C07295=1233.032,115.078,-48.574,-178.231,5.533,148.437
C07296=1233.037,114.829,-48.555,-178.233,5.532,148.437
C07297=1233.042,114.580,-48.535,-178.236,5.532,148.438
C07298=1233.046,114.331,-48.516,-178.239,5.530,148.438
C07299=1233.051,114.082,-48.497,-178.241,5.529,148.439
C07300=1233.056,113.832,-48.477,-178.244,5.529,148.439
C07301=1233.062,113.583,-48.458,-178.246,5.528,148.440
C07302=1233.066,113.334,-48.438,-178.248,5.527,148.441
C07303=1233.070,113.084,-48.419,-178.251,5.526,148.441
C07304=1233.075,112.836,-48.399,-178.254,5.525,148.442
C07305=1233.080,112.587,-48.380,-178.256,5.524,148.442
C07306=1233.085,112.337,-48.360,-178.259,5.524,148.443
C07307=1233.090,112.088,-48.341,-178.261,5.523,148.443
C07308=1233.094,111.839,-48.322,-178.264,5.521,148.444
C07309=1233.099,111.590,-48.302,-178.267,5.520,148.445
C07310=1233.104,111.341,-48.283,-178.269,5.520,148.445
C07311=1233.109,111.091,-48.263,-178.271,5.519,148.446
C07312=1233.114,110.842,-48.244,-178.274,5.518,148.446
C07313=1233.118,110.593,-48.225,-178.277,5.516,148.447
C07314=1233.124,110.344,-48.205,-178.279,5.516,148.447
C07315=1233.128,110.094,-48.186,-178.282,5.515,148.448
C07316=1233.132,109.845,-48.167,-178.284,5.514,148.448
C07317=1233.138,109.596,-48.147,-178.287,5.514,148.449
C07318=1233.143,109.347,-48.128,-178.289,5.513,148.450
C07319=1233.147,109.098,-48.110,-178.292,5.511,148.450
C07320=1233.152,108.848,-48.090,-178.295,5.511,148.451
C07321=1233.157,108.599,-48.071,-178.297,5.510,148.451
C07322=1233.162,108.350,-48.052,-178.299,5.509,148.452
C07323=1233.166,108.081,-48.031,-178.302,5.508,148.452
C07324=1233.172,107.813,-48.010,-178.305,5.507,148.453
C07325=1233.177,107.545,-47.989,-178.308,5.506,148.454
C07326=1233.183,107.276,-47.969,-178.310,5.506,148.454
C07327=1233.187,107.026,-47.949,-178.313,5.504,148.455
C07328=1233.192,106.778,-47.930,-178.316,5.503,148.455
C07329=1233.197,106.528,-47.911,-178.318,5.503,148.456
C07330=1233.201,106.280,-47.892,-178.320,5.502,148.456
C07331=1233.206,106.030,-47.873,-178.323,5.501,148.457
C07332=1233.212,105.781,-47.854,-178.326,5.500,148.458
C07333=1233.216,105.531,-47.835,-178.329,5.499,148.458
C07334=1233.221,105.283,-47.815,-178.331,5.498,148.459
C07335=1233.226,105.033,-47.796,-178.334,5.497,148.459
C07336=1233.231,104.784,-47.778,-178.336,5.497,148.460
C07337=1233.236,104.534,-47.758,-178.338,5.496,148.460
C07338=1233.240,104.286,-47.739,-178.341,5.495,148.461
C07339=1233.245,104.036,-47.720,-178.344,5.495,148.462
C07340=1233.250,103.787,-47.702,-178.346,5.493,148.462
C07341=1233.255,103.537,-47.682,-178.349,5.492,148.463
C07342=1233.260,103.289,-47.663,-178.351,5.491,148.463
C07343=1233.264,103.039,-47.644,-178.354,5.491,148.464
C07344=1233.270,102.790,-47.625,-178.356,5.490,148.464
C07345=1233.274,102.541,-47.606,-178.359,5.489,148.465
C07346=1233.279,102.292,-47.587,-178.361,5.489,148.466
C07347=1233.283,102.042,-47.569,-178.364,5.487,148.466
C07348=1233.289,101.793,-47.549,-178.367,5.486,148.467
C07349=1233.293,101.544,-47.530,-178.369,5.486,148.467
C07350=1233.298,101.294,-47.512,-178.371,5.485,148.468
C07351=1233.303,101.046,-47.493,-178.374,5.484,148.469
C07352=1233.308,100.796,-47.473,-178.377,5.483,148.469
C07353=1233.312,100.547,-47.455,-178.379,5.482,148.470
C07354=1233.317,100.297,-47.436,-178.382,5.481,148.470
C07355=1233.322,100.049,-47.417,-178.385,5.480,148.471
C07356=1233.327,99.799,-47.398,-178.387,5.480,148.472
C07357=1233.331,99.550,-47.379,-178.389,5.479,148.472
C07358=1233.336,99.301,-47.361,-178.392,5.478,148.473
C07359=1233.341,99.051,-47.342,-178.395,5.478,148.473
C07360=1233.346,98.803,-47.323,-178.397,5.477,148.474
C07361=1233.351,98.553,-47.304,-178.399,5.476,148.474
C07362=1233.355,98.304,-47.285,-178.402,5.475,148.475
C07363=1233.361,98.055,-47.267,-178.405,5.474,148.476
C07364=1233.365,97.805,-47.248,-178.407,5.473,148.476
C07365=1233.370,97.556,-47.230,-178.410,5.472,148.477
C07366=1233.375,97.307,-47.210,-178.412,5.472,148.477
C07367=1233.380,97.057,-47.192,-178.415,5.471,148.478
C07368=1233.385,96.808,-47.173,-178.417,5.470,148.478
C07369=1233.389,96.559,-47.154,-178.420,5.470,148.479
C07370=1233.394,96.310,-47.136,-178.422,5.469,148.480
C07371=1233.399,96.061,-47.117,-178.425,5.467,148.480
C07372=1233.403,95.811,-47.098,-178.428,5.467,148.481
C07373=1233.409,95.562,-47.080,-178.430,5.466,148.481
C07374=1233.413,95.313,-47.060,-178.433,5.465,148.482
C07375=1233.418,95.063,-47.042,-178.435,5.464,148.482
C07376=1233.424,94.814,-47.024,-178.438,5.464,148.483
C07377=1233.428,94.565,-47.005,-178.440,5.463,148.484
C07378=1233.433,94.315,-46.987,-178.443,5.463,148.484
C07379=1233.438,94.067,-46.968,-178.445,5.462,148.485
C07380=1233.442,93.817,-46.949,-178.448,5.461,148.485
C07381=1233.447,93.568,-46.931,-178.450,5.460,148.486
C07382=1233.453,93.319,-46.912,-178.454,5.459,148.487
C07383=1233.457,93.069,-46.894,-178.456,5.458,148.487
C07384=1233.461,92.820,-46.875,-178.458,5.457,148.488
C07385=1233.466,92.571,-46.857,-178.461,5.457,148.488
C07386=1233.472,92.322,-46.838,-178.463,5.456,148.489
C07387=1233.476,92.072,-46.819,-178.466,5.455,148.490
C07388=1233.481,91.823,-46.801,-178.468,5.455,148.490
C07389=1233.487,91.574,-46.783,-178.471,5.454,148.491
C07390=1233.491,91.324,-46.764,-178.473,5.453,148.491
C07391=1233.495,91.075,-46.746,-178.476,5.452,148.492
C07392=1233.500,90.826,-46.728,-178.478,5.452,148.493
C07393=1233.506,90.577,-46.709,-178.481,5.451,148.493
C07394=1233.510,90.327,-46.690,-178.484,5.450,148.494
C07395=1233.515,90.078,-46.672,-178.486,5.449,148.494
C07396=1233.520,89.829,-46.654,-178.489,5.448,148.495
C07397=1233.524,89.579,-46.636,-178.491,5.448,148.496
C07398=1233.530,89.330,-46.617,-178.494,5.447,148.496
C07399=1233.534,89.081,-46.599,-178.496,5.446,148.497
C07400=1233.539,88.832,-46.581,-178.499,5.445,148.497
C07401=1233.544,88.582,-46.562,-178.501,5.445,148.498
C07402=1233.549,88.333,-46.544,-178.504,5.444,148.499
C07403=1233.554,88.084,-46.525,-178.506,5.443,148.499
C07404=1233.559,87.835,-46.507,-178.509,5.443,148.500
C07405=1233.563,87.585,-46.489,-178.511,5.442,148.500
C07406=1233.568,87.336,-46.471,-178.514,5.441,148.501
C07407=1233.573,87.087,-46.453,-178.516,5.440,148.501
C07408=1233.578,86.837,-46.435,-178.519,5.440,148.502
C07409=1233.583,86.589,-46.415,-178.522,5.438,148.503
C07410=1233.588,86.339,-46.397,-178.525,5.438,148.503
C07411=1233.592,86.089,-46.379,-178.527,5.437,148.504
C07412=1233.597,85.840,-46.361,-178.529,5.436,148.504
C07413=1233.602,85.591,-46.343,-178.532,5.436,148.505
C07414=1233.607,85.342,-46.325,-178.535,5.435,148.506
C07415=1233.612,85.092,-46.307,-178.537,5.434,148.506
C07416=1233.616,84.843,-46.289,-178.539,5.433,148.507
C07417=1233.621,84.594,-46.271,-178.542,5.433,148.508
C07418=1233.627,84.344,-46.252,-178.545,5.432,148.508
C07419=1233.632,84.095,-46.234,-178.547,5.432,148.509
C07420=1233.636,83.846,-46.215,-178.550,5.431,148.509
C07421=1233.641,83.597,-46.197,-178.552,5.430,148.510
C07422=1233.646,83.347,-46.179,-178.555,5.429,148.511
C07423=1233.651,83.098,-46.161,-178.557,5.429,148.511
C07424=1233.656,82.849,-46.143,-178.560,5.428,148.512
C07425=1233.660,82.600,-46.125,-178.562,5.427,148.512
C07426=1233.665,82.350,-46.107,-178.565,5.427,148.513
C07427=1233.670,82.082,-46.088,-178.568,5.425,148.514
C07428=1233.675,81.813,-46.069,-178.570,5.425,148.514
C07429=1233.681,81.544,-46.049,-178.573,5.424,148.515
C07430=1233.686,81.276,-46.029,-178.576,5.423,148.516
C07431=1233.691,81.027,-46.011,-178.578,5.423,148.516
C07432=1233.696,80.778,-45.993,-178.581,5.422,148.517
C07433=1233.701,80.529,-45.975,-178.584,5.422,148.518
C07434=1233.706,80.279,-45.958,-178.586,5.421,148.518
C07435=1233.711,80.030,-45.940,-178.588,5.420,148.519
C07436=1233.716,79.781,-45.922,-178.591,5.420,148.519
C07437=1233.721,79.532,-45.904,-178.594,5.419,148.520
C07438=1233.726,79.282,-45.886,-178.596,5.418,148.521
C07439=1233.730,79.032,-45.868,-178.599,5.418,148.521
C07440=1233.735,78.783,-45.850,-178.601,5.417,148.522
C07441=1233.739,78.534,-45.833,-178.604,5.416,148.522
C07442=1233.744,78.285,-45.815,-178.606,5.416,148.523
C07443=1233.749,78.036,-45.797,-178.609,5.415,148.524
C07444=1233.754,77.787,-45.779,-178.611,5.414,148.524
C07445=1233.759,77.537,-45.761,-178.614,5.413,148.525
C07446=1233.764,77.288,-45.743,-178.616,5.413,148.525
C07447=1233.769,77.038,-45.725,-178.619,5.412,148.526
C07448=1233.774,76.789,-45.707,-178.621,5.412,148.527
C07449=1233.779,76.540,-45.689,-178.624,5.411,148.527
C07450=1233.784,76.290,-45.672,-178.626,5.410,148.528
C07451=1233.789,76.041,-45.654,-178.629,5.409,148.528
C07452=1233.793,75.791,-45.636,-178.631,5.409,148.529
C07453=1233.797,75.542,-45.618,-178.634,5.408,148.530
C07454=1233.803,75.293,-45.601,-178.637,5.408,148.530
C07455=1233.807,75.043,-45.583,-178.639,5.407,148.531
C07456=1233.812,74.794,-45.565,-178.641,5.406,148.532
C07457=1233.817,74.545,-45.547,-178.644,5.406,148.532
C07458=1233.823,74.295,-45.530,-178.647,5.405,148.533
C07459=1233.827,74.046,-45.512,-178.649,5.404,148.534
C07460=1233.832,73.797,-45.495,-178.652,5.404,148.534
C07461=1233.837,73.547,-45.477,-178.654,5.403,148.535
C07462=1233.842,73.298,-45.459,-178.657,5.402,148.535
C07463=1233.847,73.049,-45.441,-178.659,5.402,148.536
C07464=1233.852,72.799,-45.424,-178.662,5.401,148.537
C07465=1233.856,72.550,-45.407,-178.665,5.400,148.537
C07466=1233.861,72.301,-45.389,-178.667,5.400,148.538
C07467=1233.866,72.051,-45.372,-178.669,5.399,148.538
C07468=1233.871,71.802,-45.354,-178.672,5.398,148.539
C07469=1233.876,71.553,-45.336,-178.675,5.398,148.540
C07470=1233.880,71.304,-45.319,-178.677,5.397,148.540
C07471=1233.885,71.054,-45.301,-178.680,5.397,148.541
C07472=1233.891,70.805,-45.284,-178.683,5.396,148.542
C07473=1233.896,70.555,-45.266,-178.685,5.395,148.542
C07474=1233.900,70.306,-45.248,-178.687,5.394,148.543
C07475=1233.905,70.057,-45.231,-178.690,5.394,148.543
C07476=1233.910,69.808,-45.213,-178.693,5.393,148.544
C07477=1233.915,69.558,-45.196,-178.695,5.393,148.545
C07478=1233.919,69.309,-45.178,-178.698,5.392,148.545
C07479=1233.925,69.060,-45.162,-178.700,5.391,148.546
C07480=1233.930,68.811,-45.144,-178.703,5.390,148.546
C07481=1233.935,68.561,-45.126,-178.705,5.390,148.547
C07482=1233.939,68.312,-45.109,-178.708,5.389,148.548
C07483=1233.945,68.062,-45.092,-178.710,5.389,148.548
C07484=1233.949,67.813,-45.074,-178.713,5.388,148.549
C07485=1233.954,67.564,-45.057,-178.716,5.388,148.550
C07486=1233.959,67.314,-45.039,-178.718,5.387,148.550
C07487=1233.964,67.065,-45.022,-178.721,5.386,148.551
C07488=1233.968,66.816,-45.004,-178.723,5.385,148.552
C07489=1233.973,66.566,-44.987,-178.726,5.385,148.552
C07490=1233.978,66.317,-44.969,-178.728,5.384,148.553
C07491=1233.983,66.067,-44.952,-178.731,5.384,148.554
C07492=1233.988,65.819,-44.935,-178.734,5.383,148.554
C07493=1233.994,65.569,-44.918,-178.736,5.382,148.555
C07494=1233.998,65.320,-44.901,-178.738,5.382,148.555
C07495=1234.003,65.070,-44.883,-178.741,5.381,148.556
C07496=1234.008,64.821,-44.866,-178.743,5.381,148.557
C07497=1234.012,64.572,-44.848,-178.746,5.381,148.557
C07498=1234.018,64.322,-44.831,-178.748,5.380,148.558
C07499=1234.022,64.072,-44.814,-178.751,5.379,148.559
C07500=1234.027,63.823,-44.796,-178.754,5.379,148.559
C07501=1234.033,63.574,-44.779,-178.756,5.378,148.560
C07502=1234.037,63.325,-44.763,-178.758,5.377,148.560
C07503=1234.042,63.076,-44.745,-178.761,5.377,148.561
C07504=1234.047,62.826,-44.728,-178.764,5.376,148.562
C07505=1234.052,62.576,-44.711,-178.766,5.376,148.562
C07506=1234.057,62.327,-44.693,-178.769,5.375,148.563
C07507=1234.061,62.078,-44.676,-178.772,5.374,148.564
C07508=1234.067,61.828,-44.659,-178.774,5.374,148.564
C07509=1234.071,61.580,-44.642,-178.776,5.373,148.565
C07510=1234.077,61.330,-44.625,-178.779,5.372,148.565
C07511=1234.081,61.080,-44.608,-178.782,5.372,148.566
C07512=1234.086,60.831,-44.591,-178.784,5.371,148.567
C07513=1234.090,60.582,-44.573,-178.786,5.371,148.567
C07514=1234.096,60.333,-44.556,-178.789,5.371,148.568
C07515=1234.101,60.083,-44.540,-178.792,5.370,148.569
C07516=1234.106,59.833,-44.523,-178.794,5.370,148.569
C07517=1234.110,59.584,-44.505,-178.796,5.369,148.570
C07518=1234.115,59.335,-44.488,-178.799,5.368,148.571
C07519=1234.120,59.086,-44.472,-178.802,5.367,148.571
C07520=1234.126,58.836,-44.454,-178.804,5.367,148.572
C07521=1234.130,58.587,-44.438,-178.807,5.366,148.573
C07522=1234.135,58.337,-44.420,-178.810,5.366,148.573
C07523=1234.139,58.088,-44.403,-178.812,5.365,148.574
C07524=1234.145,57.839,-44.386,-178.815,5.365,148.575
C07525=1234.150,57.589,-44.369,-178.817,5.364,148.575
C07526=1234.155,57.340,-44.352,-178.819,5.364,148.576
C07527=1234.159,57.090,-44.335,-178.822,5.363,148.576
C07528=1234.165,56.841,-44.319,-178.824,5.363,148.577
C07529=1234.169,56.592,-44.301,-178.827,5.362,148.578
C07530=1234.174,56.343,-44.285,-178.830,5.361,148.578
C07531=1234.180,56.074,-44.266,-178.832,5.361,148.579
C07532=1234.185,55.806,-44.248,-178.835,5.360,148.580
C07533=1234.190,55.536,-44.230,-178.837,5.360,148.580
C07534=1234.196,55.269,-44.212,-178.840,5.359,148.581
C07535=1234.201,55.019,-44.195,-178.843,5.359,148.582
C07536=1234.205,54.770,-44.178,-178.845,5.358,148.582
C07537=1234.211,54.521,-44.161,-178.848,5.357,148.583
C07538=1234.215,54.271,-44.144,-178.851,5.357,148.584
C07539=1234.220,54.022,-44.128,-178.853,5.356,148.584
C07540=1234.226,53.773,-44.111,-178.856,5.356,148.585
C07541=1234.230,53.523,-44.094,-178.859,5.355,148.586
C07542=1234.234,53.274,-44.077,-178.861,5.355,148.586
C07543=1234.240,53.024,-44.060,-178.864,5.354,148.587
C07544=1234.245,52.775,-44.044,-178.865,5.354,148.587
C07545=1234.249,52.526,-44.027,-178.868,5.353,148.588
C07546=1234.254,52.276,-44.010,-178.871,5.353,148.589
C07547=1234.260,52.027,-43.993,-178.873,5.352,148.589
C07548=1234.264,51.778,-43.977,-178.876,5.352,148.590
C07549=1234.269,51.528,-43.960,-178.879,5.351,148.591
C07550=1234.275,51.278,-43.944,-178.881,5.350,148.591
C07551=1234.279,51.029,-43.927,-178.884,5.350,148.592
C07552=1234.284,50.779,-43.910,-178.886,5.349,148.593
C07553=1234.289,50.530,-43.894,-178.889,5.349,148.594
C07554=1234.294,50.281,-43.877,-178.891,5.349,148.594
C07555=1234.298,50.031,-43.860,-178.893,5.348,148.595
C07556=1234.304,49.782,-43.843,-178.896,5.347,148.595
C07557=1234.309,49.533,-43.827,-178.899,5.347,148.596
C07558=1234.313,49.283,-43.810,-178.901,5.346,148.597
C07559=1234.319,49.034,-43.793,-178.904,5.346,148.597
C07560=1234.324,48.784,-43.777,-178.906,5.345,148.598
C07561=1234.328,48.535,-43.761,-178.909,5.345,148.599
C07562=1234.333,48.286,-43.744,-178.911,5.345,148.599
C07563=1234.338,48.036,-43.728,-178.914,5.344,148.600
C07564=1234.343,47.787,-43.710,-178.916,5.344,148.601
C07565=1234.348,47.538,-43.694,-178.919,5.343,148.601
C07566=1234.353,47.288,-43.678,-178.922,5.342,148.602
C07567=1234.358,47.039,-43.662,-178.924,5.342,148.603
C07568=1234.363,46.789,-43.645,-178.927,5.341,148.603
C07569=1234.368,46.540,-43.628,-178.929,5.340,148.604
C07570=1234.373,46.291,-43.612,-178.931,5.341,148.604
C07571=1234.378,46.041,-43.596,-178.934,5.340,148.605
C07572=1234.383,45.792,-43.579,-178.937,5.339,148.606
C07573=1234.388,45.542,-43.562,-178.939,5.339,148.606
C07574=1234.392,45.293,-43.545,-178.942,5.338,148.607
C07575=1234.398,45.043,-43.530,-178.944,5.338,148.608
C07576=1234.402,44.794,-43.513,-178.947,5.337,148.608
C07577=1234.407,44.545,-43.497,-178.949,5.337,148.609
C07578=1234.412,44.296,-43.480,-178.952,5.337,148.610
C07579=1234.417,44.045,-43.464,-178.954,5.336,148.611
C07580=1234.422,43.796,-43.447,-178.957,5.336,148.611
C07581=1234.427,43.547,-43.431,-178.960,5.335,148.612
C07582=1234.432,43.297,-43.415,-178.962,5.334,148.612
C07583=1234.437,43.048,-43.398,-178.964,5.334,148.613
C07584=1234.442,42.799,-43.382,-178.967,5.334,148.614
C07585=1234.447,42.549,-43.366,-178.969,5.333,148.614
C07586=1234.452,42.300,-43.350,-178.972,5.333,148.615
C07587=1234.456,42.051,-43.333,-178.974,5.332,148.616
C07588=1234.462,41.800,-43.317,-178.977,5.332,148.616
C07589=1234.467,41.552,-43.300,-178.980,5.331,148.617
C07590=1234.471,41.302,-43.284,-178.982,5.331,148.618
C07591=1234.477,41.053,-43.268,-178.984,5.331,148.618
C07592=1234.481,40.803,-43.251,-178.987,5.330,148.619
C07593=1234.486,40.554,-43.236,-178.990,5.330,148.620
C07594=1234.491,40.304,-43.219,-178.992,5.329,148.620
C07595=1234.496,40.055,-43.204,-178.995,5.328,148.621
C07596=1234.501,39.805,-43.187,-178.998,5.328,148.622
C07597=1234.506,39.557,-43.171,-179.000,5.328,148.622
C07598=1234.511,39.307,-43.155,-179.002,5.328,148.623
C07599=1234.516,39.058,-43.138,-179.005,5.327,148.624
C07600=1234.521,38.808,-43.122,-179.007,5.326,148.624
C07601=1234.526,38.559,-43.106,-179.010,5.326,148.625
C07602=1234.530,38.309,-43.090,-179.012,5.325,148.626
C07603=1234.535,38.060,-43.074,-179.015,5.325,148.626
C07604=1234.540,37.810,-43.058,-179.017,5.325,148.627
C07605=1234.545,37.561,-43.042,-179.020,5.324,148.628
C07606=1234.550,37.311,-43.026,-179.022,5.324,148.628
C07607=1234.555,37.062,-43.009,-179.025,5.323,148.629
C07608=1234.560,36.812,-42.993,-179.028,5.322,148.630
C07609=1234.565,36.563,-42.977,-179.030,5.323,148.630
C07610=1234.570,36.314,-42.961,-179.032,5.322,148.631
C07611=1234.575,36.064,-42.945,-179.035,5.322,148.632
C07612=1234.580,35.815,-42.929,-179.038,5.321,148.632
C07613=1234.585,35.565,-42.913,-179.040,5.320,148.633
C07614=1234.590,35.316,-42.897,-179.043,5.320,148.634
C07615=1234.595,35.066,-42.881,-179.045,5.320,148.634
C07616=1234.600,34.817,-42.865,-179.048,5.320,148.635
C07617=1234.605,34.567,-42.849,-179.050,5.319,148.636
C07618=1234.610,34.318,-42.833,-179.053,5.318,148.636
C07619=1234.615,34.069,-42.817,-179.056,5.318,148.637
C07620=1234.620,33.819,-42.801,-179.058,5.317,148.638
C07621=1234.625,33.570,-42.785,-179.060,5.318,148.638
C07622=1234.629,33.320,-42.769,-179.063,5.317,148.639
C07623=1234.635,33.071,-42.754,-179.066,5.316,148.640
C07624=1234.639,32.821,-42.737,-179.068,5.316,148.640
C07625=1234.644,32.572,-42.721,-179.070,5.315,148.641
C07626=1234.650,32.323,-42.706,-179.072,5.315,148.642
C07627=1234.655,32.073,-42.690,-179.075,5.315,148.642
C07628=1234.660,31.824,-42.673,-179.078,5.314,148.643
C07629=1234.665,31.574,-42.658,-179.080,5.314,148.644
C07630=1234.669,31.325,-42.643,-179.083,5.313,148.644
C07631=1234.674,31.076,-42.626,-179.085,5.313,148.645
C07632=1234.679,30.826,-42.610,-179.088,5.313,148.646
C07633=1234.684,30.576,-42.595,-179.090,5.312,148.646
C07634=1234.690,30.327,-42.579,-179.093,5.312,148.647
C07635=1234.695,30.058,-42.562,-179.096,5.311,148.648
C07636=1234.700,29.789,-42.545,-179.099,5.311,148.649
C07637=1234.705,29.521,-42.528,-179.101,5.310,148.649
C07638=1234.711,29.253,-42.511,-179.104,5.310,148.650
C07639=1234.715,29.003,-42.495,-179.106,5.310,148.651
C07640=1234.721,28.754,-42.479,-179.109,5.309,148.651
C07641=1234.726,28.504,-42.463,-179.111,5.309,148.652
C07642=1234.731,28.254,-42.447,-179.114,5.308,148.653
C07643=1234.735,28.005,-42.432,-179.117,5.308,148.653
C07644=1234.740,27.756,-42.416,-179.119,5.308,148.654
C07645=1234.745,27.506,-42.400,-179.122,5.307,148.655
C07646=1234.751,27.257,-42.385,-179.124,5.307,148.655
C07647=1234.755,27.008,-42.370,-179.127,5.306,148.656
C07648=1234.760,26.758,-42.354,-179.129,5.306,148.657
C07649=1234.765,26.508,-42.338,-179.132,5.306,148.657
C07650=1234.771,26.259,-42.323,-179.134,5.305,148.658
C07651=1234.775,26.010,-42.306,-179.137,5.305,148.659
C07652=1234.780,25.760,-42.291,-179.139,5.304,148.659
C07653=1234.785,25.511,-42.275,-179.142,5.304,148.660
C07654=1234.791,25.261,-42.260,-179.144,5.304,148.661
C07655=1234.795,25.012,-42.244,-179.147,5.303,148.662
C07656=1234.800,24.762,-42.229,-179.149,5.303,148.662
C07657=1234.806,24.513,-42.213,-179.152,5.302,148.663
C07658=1234.810,24.263,-42.198,-179.154,5.303,148.664
C07659=1234.815,24.014,-42.182,-179.157,5.302,148.664
C07660=1234.820,23.764,-42.167,-179.159,5.302,148.665
C07661=1234.825,23.515,-42.152,-179.162,5.301,148.666
C07662=1234.830,23.265,-42.136,-179.165,5.300,148.666
C07663=1234.835,23.016,-42.120,-179.167,5.301,148.667
C07664=1234.840,22.767,-42.105,-179.169,5.300,148.668
C07665=1234.845,22.518,-42.089,-179.172,5.300,148.668
C07666=1234.850,22.268,-42.073,-179.175,5.299,148.669
C07667=1234.854,22.019,-42.058,-179.177,5.299,148.670
C07668=1234.860,21.769,-42.043,-179.179,5.299,148.670
C07669=1234.865,21.519,-42.027,-179.182,5.298,148.671
C07670=1234.870,21.269,-42.012,-179.185,5.298,148.672
C07671=1234.875,21.020,-41.996,-179.187,5.297,148.672
C07672=1234.880,20.771,-41.981,-179.190,5.297,148.673
C07673=1234.885,20.521,-41.966,-179.192,5.297,148.674
C07674=1234.890,20.271,-41.950,-179.195,5.296,148.674
C07675=1234.894,20.022,-41.935,-179.197,5.296,148.675
C07676=1234.900,19.773,-41.919,-179.200,5.296,148.676
C07677=1234.905,19.523,-41.904,-179.202,5.295,148.677
C07678=1234.910,19.274,-41.889,-179.205,5.295,148.677
C07679=1234.915,19.024,-41.873,-179.207,5.294,148.678
C07680=1234.919,18.775,-41.858,-179.210,5.295,148.679
C07681=1234.925,18.526,-41.842,-179.212,5.294,148.679
C07682=1234.930,18.276,-41.828,-179.215,5.293,148.680
C07683=1234.935,18.027,-41.812,-179.217,5.293,148.681
C07684=1234.940,17.777,-41.796,-179.220,5.293,148.681
C07685=1234.944,17.527,-41.781,-179.222,5.293,148.682
C07686=1234.950,17.278,-41.766,-179.225,5.292,148.683
C07687=1234.954,17.029,-41.751,-179.227,5.292,148.683
C07688=1234.960,16.780,-41.735,-179.230,5.292,148.684
C07689=1234.964,16.529,-41.721,-179.232,5.291,148.685
C07690=1234.970,16.280,-41.705,-179.235,5.291,148.685
C07691=1234.974,16.031,-41.690,-179.238,5.290,148.686
C07692=1234.980,15.781,-41.674,-179.240,5.290,148.687
C07693=1234.984,15.532,-41.659,-179.242,5.290,148.687
C07694=1234.990,15.282,-41.645,-179.245,5.289,148.688
C07695=1234.994,15.032,-41.629,-179.248,5.289,148.689
C07696=1234.999,14.783,-41.614,-179.250,5.289,148.690
C07697=1235.004,14.534,-41.599,-179.252,5.289,148.690
C07698=1235.010,14.284,-41.584,-179.255,5.288,148.691
C07699=1235.014,14.035,-41.569,-179.258,5.287,148.692
C07700=1235.020,13.785,-41.553,-179.260,5.288,148.692
C07701=1235.024,13.536,-41.538,-179.262,5.287,148.693
C07702=1235.030,13.286,-41.523,-179.265,5.287,148.694
C07703=1235.034,13.036,-41.508,-179.268,5.286,148.694
C07704=1235.039,12.787,-41.493,-179.270,5.286,148.695
C07705=1235.044,12.538,-41.477,-179.272,5.286,148.696
C07706=1235.049,12.288,-41.463,-179.275,5.285,148.696
C07707=1235.055,12.039,-41.447,-179.278,5.285,148.697
C07708=1235.059,11.790,-41.432,-179.280,5.285,148.698
C07709=1235.065,11.540,-41.418,-179.282,5.284,148.698
C07710=1235.069,11.291,-41.403,-179.285,5.284,148.699
C07711=1235.074,11.042,-41.388,-179.287,5.284,148.700
C07712=1235.079,10.791,-41.372,-179.290,5.284,148.700
C07713=1235.084,10.542,-41.357,-179.292,5.283,148.701
C07714=1235.090,10.292,-41.343,-179.295,5.283,148.702
C07715=1235.094,10.043,-41.328,-179.297,5.283,148.703
C07716=1235.099,9.794,-41.313,-179.300,5.282,148.703
C07717=1235.105,9.543,-41.298,-179.302,5.282,148.704
C07718=1235.109,9.294,-41.283,-179.305,5.281,148.705
C07719=1235.114,9.045,-41.268,-179.307,5.281,148.705
C07720=1235.120,8.795,-41.253,-179.310,5.281,148.706
C07721=1235.124,8.546,-41.238,-179.312,5.280,148.707
C07722=1235.130,8.296,-41.223,-179.314,5.281,148.707
C07723=1235.135,8.047,-41.208,-179.317,5.280,148.708
C07724=1235.140,7.797,-41.194,-179.320,5.280,148.709
C07725=1235.145,7.548,-41.178,-179.322,5.279,148.709
C07726=1235.150,7.298,-41.164,-179.325,5.279,148.710
C07727=1235.154,7.049,-41.149,-179.327,5.279,148.711
C07728=1235.159,6.799,-41.135,-179.330,5.279,148.712
C07729=1235.164,6.549,-41.119,-179.333,5.278,148.712
C07730=1235.169,6.300,-41.104,-179.335,5.278,148.713
C07731=1235.174,6.051,-41.089,-179.338,5.278,148.714
C07732=1235.180,5.801,-41.074,-179.340,5.277,148.714
C07733=1235.184,5.551,-41.059,-179.342,5.278,148.715
C07734=1235.189,5.302,-41.045,-179.345,5.277,148.716
C07735=1235.194,5.053,-41.030,-179.348,5.276,148.716
C07736=1235.199,4.803,-41.015,-179.350,5.277,148.717
C07737=1235.204,4.554,-41.000,-179.352,5.276,148.718
C07738=1235.209,4.304,-40.986,-179.355,5.276,148.719
C07739=1235.215,4.035,-40.970,-179.358,5.275,148.719
C07740=1235.220,3.766,-40.954,-179.360,5.275,148.720
C07741=1235.226,3.498,-40.939,-179.363,5.275,148.721
C07742=1235.232,3.229,-40.922,-179.366,5.275,148.722
C07743=1235.236,2.980,-40.907,-179.368,5.274,148.722
C07744=1235.241,2.730,-40.893,-179.371,5.274,148.723
C07745=1235.246,2.480,-40.879,-179.373,5.274,148.724
C07746=1235.251,2.231,-40.864,-179.376,5.273,148.724
C07747=1235.257,1.981,-40.849,-179.378,5.273,148.725
C07748=1235.262,1.731,-40.835,-179.380,5.273,148.726
C07749=1235.266,1.482,-40.820,-179.383,5.273,148.726
C07750=1235.271,1.233,-40.805,-179.386,5.272,148.727
C07751=1235.276,0.983,-40.791,-179.388,5.272,148.728
C07752=1235.281,0.733,-40.776,-179.390,5.272,148.728
C07753=1235.286,0.484,-40.761,-179.393,5.271,148.729
C07754=1235.291,0.234,-40.747,-179.396,5.271,148.730
C07755=1235.296,-0.015,-40.732,-179.398,5.271,148.730
C07756=1235.301,-0.265,-40.718,-179.400,5.270,148.731
C07757=1235.306,-0.514,-40.703,-179.403,5.270,148.732
C07758=1235.311,-0.764,-40.688,-179.406,5.271,148.733
C07759=1235.316,-1.014,-40.674,-179.408,5.270,148.733
C07760=1235.322,-1.263,-40.660,-179.411,5.270,148.734
C07761=1235.327,-1.512,-40.645,-179.413,5.270,148.735
C07762=1235.331,-1.761,-40.630,-179.416,5.269,148.736
C07763=1235.336,-2.011,-40.616,-179.418,5.269,148.736
C07764=1235.341,-2.261,-40.602,-179.421,5.268,148.737
C07765=1235.346,-2.511,-40.588,-179.423,5.269,148.738
C07766=1235.352,-2.760,-40.572,-179.426,5.268,148.738
C07767=1235.357,-3.010,-40.558,-179.428,5.267,148.739
C07768=1235.362,-3.259,-40.543,-179.431,5.268,148.740
C07769=1235.367,-3.509,-40.529,-179.433,5.267,148.740
C07770=1235.372,-3.758,-40.515,-179.436,5.267,148.741
C07771=1235.377,-4.007,-40.500,-179.438,5.267,148.742
C07772=1235.382,-4.257,-40.486,-179.441,5.266,148.742
C07773=1235.387,-4.507,-40.472,-179.443,5.266,148.743
C07774=1235.392,-4.756,-40.457,-179.445,5.266,148.744
C07775=1235.397,-5.006,-40.443,-179.448,5.266,148.745
C07776=1235.402,-5.256,-40.429,-179.451,5.265,148.745
C07777=1235.407,-5.504,-40.414,-179.453,5.265,148.746
C07778=1235.412,-5.754,-40.400,-179.455,5.265,148.747
C07779=1235.417,-6.004,-40.386,-179.458,5.264,148.747
C07780=1235.422,-6.253,-40.371,-179.461,5.265,148.748
C07781=1235.427,-6.503,-40.357,-179.463,5.264,148.749
C07782=1235.432,-6.753,-40.343,-179.466,5.264,148.750
C07783=1235.437,-7.002,-40.329,-179.468,5.264,148.750
C07784=1235.442,-7.251,-40.315,-179.471,5.264,148.751
C07785=1235.447,-7.501,-40.300,-179.473,5.263,148.752
C07786=1235.452,-7.750,-40.285,-179.475,5.263,148.752
C07787=1235.457,-8.000,-40.271,-179.478,5.263,148.753
C07788=1235.462,-8.250,-40.257,-179.481,5.262,148.754
C07789=1235.467,-8.499,-40.243,-179.483,5.263,148.754
C07790=1235.472,-8.748,-40.229,-179.485,5.262,148.755
C07791=1235.477,-8.998,-40.214,-179.488,5.262,148.756
C07792=1235.482,-9.248,-40.200,-179.490,5.262,148.757
C07793=1235.487,-9.497,-40.186,-179.493,5.261,148.757
C07794=1235.492,-9.747,-40.172,-179.495,5.261,148.758
C07795=1235.497,-9.996,-40.158,-179.498,5.261,148.759
C07796=1235.502,-10.246,-40.143,-179.500,5.261,148.759
C07797=1235.507,-10.496,-40.129,-179.503,5.260,148.760
C07798=1235.512,-10.745,-40.115,-179.505,5.260,148.761
C07799=1235.517,-10.995,-40.101,-179.508,5.260,148.762
C07800=1235.523,-11.244,-40.087,-179.511,5.260,148.762
C07801=1235.528,-11.494,-40.072,-179.513,5.260,148.763
C07802=1235.533,-11.743,-40.058,-179.515,5.259,148.764
C07803=1235.537,-11.993,-40.044,-179.518,5.259,148.764
C07804=1235.543,-12.242,-40.030,-179.520,5.259,148.765
C07805=1235.548,-12.492,-40.017,-179.523,5.259,148.766
C07806=1235.553,-12.742,-40.003,-179.526,5.258,148.766
C07807=1235.558,-12.992,-39.988,-179.528,5.259,148.767
C07808=1235.563,-13.241,-39.974,-179.530,5.258,148.768
C07809=1235.568,-13.490,-39.960,-179.533,5.257,148.769
C07810=1235.573,-13.740,-39.946,-179.535,5.258,148.769
C07811=1235.578,-13.990,-39.932,-179.538,5.257,148.770
C07812=1235.583,-14.238,-39.918,-179.540,5.257,148.771
C07813=1235.588,-14.488,-39.904,-179.542,5.257,148.771
C07814=1235.593,-14.738,-39.890,-179.545,5.256,148.772
C07815=1235.598,-14.988,-39.876,-179.547,5.257,148.773
C07816=1235.604,-15.237,-39.862,-179.550,5.257,148.774
C07817=1235.609,-15.487,-39.848,-179.553,5.256,148.774
C07818=1235.613,-15.736,-39.834,-179.555,5.256,148.775
C07819=1235.618,-15.985,-39.820,-179.558,5.256,148.776
C07820=1235.623,-16.235,-39.806,-179.560,5.255,148.776
C07821=1235.629,-16.485,-39.793,-179.562,5.256,148.777
C07822=1235.634,-16.734,-39.779,-179.565,5.255,148.778
C07823=1235.638,-16.984,-39.765,-179.568,5.255,148.778
C07824=1235.643,-17.233,-39.751,-179.570,5.255,148.779
C07825=1235.649,-17.484,-39.737,-179.572,5.254,148.780
C07826=1235.654,-17.733,-39.723,-179.575,5.254,148.781
C07827=1235.659,-17.983,-39.709,-179.577,5.254,148.781
C07828=1235.663,-18.232,-39.695,-179.580,5.254,148.782
C07829=1235.669,-18.481,-39.681,-179.582,5.254,148.783
C07830=1235.674,-18.731,-39.668,-179.585,5.253,148.783
C07831=1235.679,-18.981,-39.654,-179.587,5.253,148.784
C07832=1235.684,-19.230,-39.640,-179.590,5.254,148.785
C07833=1235.689,-19.480,-39.627,-179.592,5.253,148.786
C07834=1235.694,-19.730,-39.612,-179.595,5.253,148.786
C07835=1235.700,-19.979,-39.598,-179.597,5.253,148.787
C07836=1235.704,-20.228,-39.585,-179.600,5.252,148.788
C07837=1235.709,-20.478,-39.571,-179.602,5.253,148.788
C07838=1235.715,-20.727,-39.557,-179.605,5.252,148.789
C07839=1235.720,-20.977,-39.543,-179.607,5.252,148.790
C07840=1235.725,-21.226,-39.530,-179.609,5.252,148.791
C07841=1235.730,-21.476,-39.516,-179.612,5.251,148.791
C07842=1235.735,-21.726,-39.502,-179.615,5.251,148.792
C07843=1235.741,-21.995,-39.487,-179.617,5.251,148.793
C07844=1235.746,-22.264,-39.474,-179.620,5.251,148.794
C07845=1235.751,-22.534,-39.459,-179.623,5.250,148.794
C07846=1235.757,-22.803,-39.444,-179.625,5.250,148.795
C07847=1235.762,-23.052,-39.430,-179.627,5.250,148.796
C07848=1235.766,-23.302,-39.416,-179.630,5.250,148.797
C07849=1235.772,-23.552,-39.402,-179.633,5.250,148.797
C07850=1235.777,-23.801,-39.388,-179.635,5.250,148.798
C07851=1235.782,-24.051,-39.376,-179.638,5.249,148.799
C07852=1235.787,-24.300,-39.362,-179.640,5.250,148.799
C07853=1235.793,-24.550,-39.348,-179.643,5.249,148.800
C07854=1235.797,-24.800,-39.334,-179.645,5.249,148.801
C07855=1235.802,-25.049,-39.320,-179.647,5.249,148.801
C07856=1235.807,-25.299,-39.307,-179.650,5.248,148.802
C07857=1235.812,-25.548,-39.294,-179.652,5.249,148.803
C07858=1235.818,-25.798,-39.280,-179.655,5.248,148.804
C07859=1235.822,-26.047,-39.267,-179.657,5.248,148.804
C07860=1235.828,-26.297,-39.253,-179.660,5.248,148.805
C07861=1235.832,-26.546,-39.239,-179.662,5.248,148.806
C07862=1235.838,-26.796,-39.226,-179.665,5.247,148.806
C07863=1235.843,-27.046,-39.212,-179.667,5.248,148.807
C07864=1235.848,-27.295,-39.199,-179.670,5.247,148.808
C07865=1235.853,-27.545,-39.185,-179.672,5.247,148.809
C07866=1235.858,-27.794,-39.173,-179.675,5.247,148.809
C07867=1235.863,-28.044,-39.158,-179.677,5.246,148.810
C07868=1235.868,-28.293,-39.146,-179.680,5.247,148.811
C07869=1235.873,-28.543,-39.131,-179.682,5.246,148.811
C07870=1235.878,-28.793,-39.118,-179.684,5.247,148.812
C07871=1235.883,-29.043,-39.105,-179.687,5.246,148.813
C07872=1235.888,-29.292,-39.091,-179.690,5.246,148.814
C07873=1235.893,-29.542,-39.078,-179.692,5.246,148.814
C07874=1235.898,-29.791,-39.064,-179.694,5.245,148.815
C07875=1235.904,-30.041,-39.051,-179.696,5.246,148.816
C07876=1235.908,-30.290,-39.037,-179.699,5.245,148.816
C07877=1235.914,-30.540,-39.025,-179.702,5.245,148.817
C07878=1235.919,-30.790,-39.011,-179.704,5.245,148.818
C07879=1235.924,-31.039,-38.998,-179.707,5.245,148.819
C07880=1235.929,-31.289,-38.984,-179.709,5.245,148.819
C07881=1235.934,-31.538,-38.972,-179.712,5.245,148.820
C07882=1235.939,-31.788,-38.957,-179.714,5.244,148.821
C07883=1235.944,-32.037,-38.945,-179.717,5.244,148.821
C07884=1235.949,-32.288,-38.931,-179.719,5.244,148.822
C07885=1235.954,-32.536,-38.918,-179.721,5.244,148.823
C07886=1235.959,-32.787,-38.904,-179.724,5.244,148.824
C07887=1235.965,-33.036,-38.892,-179.727,5.243,148.824
C07888=1235.969,-33.285,-38.878,-179.729,5.244,148.825
C07889=1235.975,-33.535,-38.865,-179.731,5.243,148.826
C07890=1235.980,-33.784,-38.852,-179.733,5.243,148.826
C07891=1235.985,-34.034,-38.838,-179.736,5.243,148.827
C07892=1235.990,-34.283,-38.825,-179.739,5.243,148.828
C07893=1235.995,-34.534,-38.812,-179.741,5.243,148.829
C07894=1236.000,-34.783,-38.799,-179.744,5.242,148.829
C07895=1236.005,-35.033,-38.785,-179.746,5.243,148.830
C07896=1236.010,-35.282,-38.772,-179.749,5.242,148.831
C07897=1236.015,-35.532,-38.759,-179.751,5.243,148.831
C07898=1236.021,-35.782,-38.746,-179.753,5.242,148.832
C07899=1236.026,-36.030,-38.733,-179.756,5.242,148.833
C07900=1236.031,-36.281,-38.719,-179.758,5.242,148.834
C07901=1236.036,-36.530,-38.707,-179.761,5.241,148.834
C07902=1236.040,-36.780,-38.694,-179.763,5.242,148.835
C07903=1236.046,-37.030,-38.680,-179.766,5.241,148.836
C07904=1236.051,-37.278,-38.667,-179.768,5.241,148.836
C07905=1236.056,-37.528,-38.654,-179.770,5.241,148.837
C07906=1236.062,-37.778,-38.641,-179.774,5.241,148.838
C07907=1236.066,-38.028,-38.628,-179.776,5.241,148.839
C07908=1236.072,-38.278,-38.615,-179.778,5.241,148.839
C07909=1236.077,-38.527,-38.602,-179.780,5.241,148.840
C07910=1236.081,-38.776,-38.588,-179.783,5.240,148.841
C07911=1236.087,-39.026,-38.575,-179.786,5.240,148.841
C07912=1236.092,-39.276,-38.562,-179.788,5.240,148.842
C07913=1236.097,-39.525,-38.550,-179.790,5.240,148.843
C07914=1236.103,-39.775,-38.537,-179.793,5.240,148.844
C07915=1236.107,-40.025,-38.524,-179.795,5.240,148.844
C07916=1236.112,-40.274,-38.511,-179.798,5.239,148.845
C07917=1236.117,-40.524,-38.498,-179.800,5.239,148.846
C07918=1236.122,-40.773,-38.484,-179.803,5.239,148.846
C07919=1236.127,-41.023,-38.471,-179.805,5.239,148.847
C07920=1236.132,-41.273,-38.459,-179.808,5.239,148.848
C07921=1236.138,-41.522,-38.445,-179.810,5.239,148.849
C07922=1236.143,-41.772,-38.433,-179.813,5.239,148.849
C07923=1236.148,-42.022,-38.420,-179.815,5.238,148.850
C07924=1236.153,-42.271,-38.407,-179.817,5.239,148.851
C07925=1236.158,-42.521,-38.394,-179.820,5.238,148.852
C07926=1236.163,-42.771,-38.381,-179.822,5.239,148.852
C07927=1236.168,-43.020,-38.368,-179.825,5.238,148.853
C07928=1236.173,-43.269,-38.356,-179.827,5.238,148.854
C07929=1236.179,-43.520,-38.342,-179.830,5.238,148.854
C07930=1236.184,-43.769,-38.330,-179.832,5.237,148.855
C07931=1236.189,-44.018,-38.317,-179.834,5.238,148.856
C07932=1236.193,-44.268,-38.304,-179.837,5.237,148.856
C07933=1236.199,-44.518,-38.291,-179.839,5.238,148.857
C07934=1236.204,-44.767,-38.278,-179.842,5.237,148.858
C07935=1236.209,-45.017,-38.265,-179.844,5.238,148.859
C07936=1236.214,-45.267,-38.253,-179.847,5.237,148.859
C07937=1236.219,-45.516,-38.240,-179.849,5.238,148.860
C07938=1236.224,-45.766,-38.227,-179.852,5.237,148.861
C07939=1236.229,-46.016,-38.214,-179.854,5.237,148.862
C07940=1236.235,-46.265,-38.201,-179.856,5.237,148.862
C07941=1236.240,-46.514,-38.189,-179.859,5.236,148.863
C07942=1236.244,-46.764,-38.176,-179.861,5.237,148.864
C07943=1236.250,-47.014,-38.164,-179.864,5.236,148.864
C07944=1236.255,-47.264,-38.151,-179.866,5.237,148.865
C07945=1236.261,-47.513,-38.138,-179.869,5.236,148.866
C07946=1236.265,-47.763,-38.125,-179.871,5.236,148.866
C07947=1236.271,-48.032,-38.112,-179.874,5.236,148.867
C07948=1236.276,-48.302,-38.098,-179.877,5.236,148.868
C07949=1236.281,-48.572,-38.084,-179.879,5.235,148.869
C07950=1236.288,-48.841,-38.070,-179.882,5.236,148.870
C07951=1236.292,-49.091,-38.057,-179.884,5.235,148.870
C07952=1236.298,-49.341,-38.045,-179.887,5.236,148.871
C07953=1236.303,-49.590,-38.032,-179.889,5.235,148.872
C07954=1236.308,-49.840,-38.020,-179.891,5.236,148.873
C07955=1236.313,-50.090,-38.007,-179.894,5.235,148.873
C07956=1236.318,-50.339,-37.994,-179.897,5.235,148.874
C07957=1236.323,-50.589,-37.982,-179.899,5.235,148.875
C07958=1236.328,-50.838,-37.970,-179.901,5.234,148.875
C07959=1236.333,-51.088,-37.957,-179.903,5.235,148.876
C07960=1236.339,-51.338,-37.944,-179.906,5.234,148.877
C07961=1236.344,-51.587,-37.931,-179.908,5.235,148.877
C07962=1236.349,-51.837,-37.919,-179.911,5.234,148.878
C07963=1236.354,-52.087,-37.907,-179.913,5.235,148.879
C07964=1236.359,-52.337,-37.894,-179.916,5.234,148.880
C07965=1236.364,-52.586,-37.881,-179.918,5.235,148.881
C07966=1236.369,-52.836,-37.869,-179.921,5.234,148.881
C07967=1236.374,-53.085,-37.857,-179.924,5.234,148.882
C07968=1236.379,-53.335,-37.844,-179.926,5.234,148.883
C07969=1236.384,-53.585,-37.831,-179.928,5.233,148.883
C07970=1236.390,-53.834,-37.819,-179.930,5.234,148.884
C07971=1236.395,-54.084,-37.806,-179.933,5.233,148.885
C07972=1236.400,-54.333,-37.794,-179.935,5.234,148.885
C07973=1236.405,-54.583,-37.782,-179.938,5.233,148.886
C07974=1236.410,-54.833,-37.769,-179.940,5.233,148.887
C07975=1236.415,-55.082,-37.756,-179.943,5.233,148.888
C07976=1236.420,-55.332,-37.745,-179.945,5.233,148.888
C07977=1236.425,-55.582,-37.732,-179.948,5.233,148.889
C07978=1236.431,-55.831,-37.719,-179.950,5.233,148.890
C07979=1236.436,-56.081,-37.707,-179.953,5.233,148.891
C07980=1236.441,-56.331,-37.694,-179.955,5.233,148.891
C07981=1236.446,-56.580,-37.682,-179.957,5.233,148.892
C07982=1236.451,-56.830,-37.670,-179.960,5.232,148.893
C07983=1236.456,-57.079,-37.657,-179.962,5.233,148.893
C07984=1236.461,-57.329,-37.645,-179.965,5.232,148.894
C07985=1236.467,-57.579,-37.633,-179.967,5.233,148.895
C07986=1236.471,-57.829,-37.620,-179.969,5.232,148.896
C07987=1236.476,-58.078,-37.609,-179.972,5.232,148.896
C07988=1236.481,-58.328,-37.596,-179.974,5.232,148.897
C07989=1236.486,-58.577,-37.583,-179.976,5.232,148.898
C07990=1236.492,-58.827,-37.572,-179.979,5.232,148.898
C07991=1236.497,-59.076,-37.559,-179.982,5.231,148.899
C07992=1236.502,-59.326,-37.547,-179.984,5.232,148.900
C07993=1236.507,-59.575,-37.534,-179.987,5.231,148.901
C07994=1236.512,-59.826,-37.522,-179.989,5.232,148.901
C07995=1236.517,-60.075,-37.510,-179.992,5.231,148.902
C07996=1236.523,-60.325,-37.498,-179.994,5.232,148.903
C07997=1236.528,-60.575,-37.485,-179.996,5.231,148.904
C07998=1236.533,-60.824,-37.474,-179.999,5.231,148.904
C07999=1236.538,-61.074,-37.461,179.999,5.231,148.905
C08000=1236.543,-61.324,-37.449,179.997,5.231,148.906
C08001=1236.548,-61.573,-37.437,179.994,5.231,148.906
C08002=1236.554,-61.823,-37.425,179.992,5.231,148.907
C08003=1236.559,-62.072,-37.412,179.989,5.231,148.908
C08004=1236.564,-62.322,-37.400,179.987,5.231,148.908
C08005=1236.569,-62.571,-37.388,179.985,5.231,148.909
C08006=1236.573,-62.822,-37.376,179.982,5.231,148.910
C08007=1236.579,-63.071,-37.364,179.980,5.230,148.911
C08008=1236.584,-63.321,-37.352,179.978,5.231,148.911
C08009=1236.589,-63.570,-37.339,179.975,5.231,148.912
C08010=1236.594,-63.820,-37.327,179.972,5.230,148.913
C08011=1236.599,-64.070,-37.316,179.970,5.230,148.914
C08012=1236.604,-64.319,-37.303,179.967,5.230,148.914
C08013=1236.610,-64.569,-37.291,179.965,5.230,148.915
C08014=1236.615,-64.818,-37.279,179.962,5.230,148.916
C08015=1236.620,-65.068,-37.267,179.960,5.230,148.916
C08016=1236.625,-65.318,-37.256,179.958,5.230,148.917
C08017=1236.630,-65.567,-37.243,179.955,5.230,148.918
C08018=1236.636,-65.817,-37.231,179.953,5.230,148.919
C08019=1236.641,-66.067,-37.219,179.951,5.230,148.919
C08020=1236.646,-66.317,-37.207,179.948,5.229,148.920
C08021=1236.651,-66.566,-37.195,179.946,5.230,148.921
C08022=1236.656,-66.815,-37.183,179.943,5.229,148.921
C08023=1236.661,-67.065,-37.171,179.941,5.230,148.922
C08024=1236.667,-67.315,-37.159,179.939,5.229,148.923
C08025=1236.671,-67.564,-37.147,179.936,5.229,148.924
C08026=1236.677,-67.814,-37.135,179.934,5.229,148.924
C08027=1236.682,-68.064,-37.123,179.931,5.230,148.925
C08028=1236.687,-68.314,-37.111,179.929,5.229,148.926
C08029=1236.692,-68.563,-37.099,179.926,5.230,148.927
C08030=1236.697,-68.813,-37.087,179.924,5.229,148.927
C08031=1236.703,-69.063,-37.076,179.922,5.229,148.928
C08032=1236.707,-69.312,-37.064,179.919,5.229,148.929
C08033=1236.712,-69.562,-37.052,179.917,5.229,148.929
C08034=1236.718,-69.812,-37.040,179.914,5.229,148.930
C08035=1236.723,-70.062,-37.028,179.912,5.229,148.931
C08036=1236.728,-70.311,-37.016,179.909,5.229,148.932
C08037=1236.733,-70.561,-37.004,179.907,5.229,148.932
C08038=1236.739,-70.811,-36.992,179.905,5.228,148.933
C08039=1236.743,-71.060,-36.981,179.903,5.229,148.934
C08040=1236.748,-71.310,-36.968,179.900,5.228,148.934
C08041=1236.754,-71.560,-36.956,179.898,5.229,148.935
C08042=1236.759,-71.809,-36.945,179.895,5.228,148.936
C08043=1236.764,-72.059,-36.933,179.893,5.229,148.937
C08044=1236.769,-72.309,-36.921,179.890,5.228,148.937
C08045=1236.774,-72.557,-36.910,179.888,5.228,148.938
C08046=1236.780,-72.807,-36.898,179.886,5.228,148.939
C08047=1236.785,-73.057,-36.886,179.883,5.228,148.940
C08048=1236.790,-73.307,-36.875,179.880,5.228,148.940
C08049=1236.795,-73.557,-36.863,179.878,5.228,148.941
C08050=1236.801,-73.807,-36.851,179.876,5.228,148.942
C08051=1236.806,-74.077,-36.838,179.873,5.228,148.942
C08052=1236.812,-74.347,-36.825,179.871,5.228,148.943
C08053=1236.817,-74.617,-36.812,179.868,5.228,148.944
C08054=1236.823,-74.888,-36.800,179.865,5.227,148.945
C08055=1236.828,-75.136,-36.788,179.863,5.228,148.945
C08056=1236.833,-75.386,-36.776,179.860,5.227,148.946
C08057=1236.838,-75.636,-36.765,179.858,5.228,148.947
C08058=1236.843,-75.886,-36.753,179.856,5.227,148.948
C08059=1236.848,-76.136,-36.742,179.853,5.227,148.948
C08060=1236.854,-76.385,-36.730,179.851,5.227,148.949
C08061=1236.859,-76.635,-36.718,179.849,5.227,148.950
C08062=1236.864,-76.885,-36.707,179.846,5.227,148.950
C08063=1236.869,-77.135,-36.695,179.844,5.227,148.951
C08064=1236.874,-77.384,-36.684,179.841,5.227,148.952
C08065=1236.880,-77.634,-36.672,179.839,5.227,148.953
C08066=1236.885,-77.883,-36.661,179.836,5.227,148.953
C08067=1236.890,-78.133,-36.649,179.834,5.227,148.954
C08068=1236.895,-78.383,-36.638,179.832,5.226,148.955
C08069=1236.900,-78.633,-36.626,179.830,5.227,148.955
C08070=1236.905,-78.883,-36.615,179.827,5.228,148.956
C08071=1236.911,-79.132,-36.603,179.824,5.227,148.957
C08072=1236.916,-79.382,-36.591,179.822,5.227,148.958
C08073=1236.921,-79.631,-36.580,179.820,5.227,148.958
C08074=1236.926,-79.881,-36.568,179.818,5.227,148.959
C08075=1236.931,-80.131,-36.557,179.815,5.227,148.960
C08076=1236.937,-80.381,-36.545,179.813,5.227,148.961
C08077=1236.942,-80.630,-36.534,179.810,5.227,148.961
C08078=1236.946,-80.879,-36.523,179.808,5.227,148.962
C08079=1236.952,-81.129,-36.511,179.805,5.227,148.963
C08080=1236.957,-81.379,-36.499,179.803,5.227,148.963
C08081=1236.962,-81.629,-36.488,179.801,5.226,148.964
C08082=1236.967,-81.878,-36.477,179.798,5.227,148.965
C08083=1236.973,-82.128,-36.465,179.796,5.226,148.966
C08084=1236.977,-82.377,-36.453,179.794,5.227,148.966
C08085=1236.983,-82.627,-36.442,179.791,5.226,148.967
C08086=1236.988,-82.878,-36.431,179.789,5.227,148.968
C08087=1236.993,-83.128,-36.419,179.786,5.226,148.968
C08088=1236.999,-83.376,-36.408,179.784,5.226,148.969
C08089=1237.003,-83.626,-36.397,179.782,5.226,148.970
C08090=1237.009,-83.876,-36.385,179.779,5.226,148.971
C08091=1237.013,-84.126,-36.374,179.777,5.226,148.971
C08092=1237.019,-84.375,-36.362,179.775,5.226,148.972
C08093=1237.024,-84.625,-36.351,179.772,5.226,148.973
C08094=1237.029,-84.875,-36.340,179.770,5.226,148.973
C08095=1237.035,-85.125,-36.328,179.767,5.226,148.974
C08096=1237.039,-85.374,-36.317,179.765,5.226,148.975
C08097=1237.045,-85.624,-36.306,179.762,5.225,148.976
C08098=1237.050,-85.873,-36.294,179.760,5.226,148.976
C08099=1237.055,-86.123,-36.284,179.758,5.225,148.977
C08100=1237.060,-86.373,-36.272,179.756,5.226,148.978
C08101=1237.066,-86.622,-36.261,179.753,5.225,148.978
C08102=1237.070,-86.872,-36.250,179.751,5.226,148.979
C08103=1237.076,-87.122,-36.238,179.748,5.226,148.980
C08104=1237.081,-87.372,-36.227,179.746,5.226,148.981
C08105=1237.086,-87.621,-36.216,179.743,5.225,148.981
C08106=1237.092,-87.871,-36.204,179.741,5.226,148.982
C08107=1237.096,-88.121,-36.193,179.738,5.225,148.983
C08108=1237.102,-88.370,-36.183,179.736,5.226,148.984
C08109=1237.107,-88.620,-36.171,179.734,5.226,148.984
C08110=1237.112,-88.870,-36.160,179.731,5.226,148.985
C08111=1237.117,-89.119,-36.148,179.729,5.226,148.986
C08112=1237.123,-89.369,-36.138,179.726,5.225,148.986
C08113=1237.128,-89.619,-36.126,179.724,5.226,148.987
C08114=1237.132,-89.868,-36.115,179.722,5.225,148.988
C08115=1237.139,-90.118,-36.104,179.720,5.226,148.989
C08116=1237.143,-90.368,-36.093,179.717,5.225,148.989
C08117=1237.148,-90.618,-36.082,179.715,5.226,148.990
C08118=1237.153,-90.868,-36.071,179.712,5.225,148.991
C08119=1237.159,-91.117,-36.060,179.710,5.225,148.991
C08120=1237.164,-91.367,-36.048,179.707,5.225,148.992
C08121=1237.169,-91.617,-36.038,179.705,5.225,148.993
C08122=1237.174,-91.866,-36.027,179.703,5.225,148.994
C08123=1237.180,-92.116,-36.015,179.701,5.225,148.994
C08124=1237.185,-92.366,-36.004,179.698,5.225,148.995
C08125=1237.190,-92.615,-35.993,179.696,5.225,148.996
C08126=1237.195,-92.865,-35.982,179.693,5.225,148.996
C08127=1237.200,-93.115,-35.971,179.691,5.225,148.997
C08128=1237.206,-93.364,-35.960,179.688,5.225,148.998
C08129=1237.211,-93.614,-35.949,179.686,5.225,148.999
C08130=1237.215,-93.864,-35.938,179.684,5.225,148.999
C08131=1237.221,-94.113,-35.927,179.682,5.225,149.000
C08132=1237.226,-94.363,-35.916,179.679,5.225,149.001
C08133=1237.231,-94.613,-35.905,179.677,5.225,149.001
C08134=1237.237,-94.863,-35.895,179.675,5.225,149.002
C08135=1237.241,-95.112,-35.883,179.672,5.225,149.003
C08136=1237.248,-95.362,-35.873,179.670,5.225,149.003
C08137=1237.252,-95.612,-35.861,179.667,5.224,149.004
C08138=1237.257,-95.862,-35.851,179.665,5.225,149.005
C08139=1237.263,-96.111,-35.840,179.662,5.224,149.006
C08140=1237.267,-96.360,-35.828,179.660,5.225,149.006
C08141=1237.273,-96.611,-35.817,179.658,5.224,149.007
C08142=1237.278,-96.860,-35.806,179.656,5.225,149.008
C08143=1237.283,-97.110,-35.796,179.653,5.224,149.008
C08144=1237.289,-97.359,-35.785,179.651,5.225,149.009
C08145=1237.294,-97.609,-35.774,179.649,5.225,149.010
C08146=1237.299,-97.860,-35.764,179.646,5.224,149.011
C08147=1237.304,-98.108,-35.753,179.644,5.225,149.011
C08148=1237.310,-98.359,-35.742,179.641,5.224,149.012
C08149=1237.315,-98.608,-35.731,179.639,5.225,149.013
C08150=1237.320,-98.858,-35.720,179.636,5.224,149.013
C08151=1237.325,-99.107,-35.709,179.634,5.225,149.014
C08152=1237.330,-99.357,-35.699,179.632,5.224,149.015
C08153=1237.335,-99.607,-35.687,179.630,5.225,149.016
C08154=1237.340,-99.857,-35.677,179.627,5.224,149.016
C08155=1237.346,-100.128,-35.665,179.625,5.224,149.017
C08156=1237.352,-100.399,-35.653,179.622,5.224,149.018
C08157=1237.357,-100.669,-35.642,179.620,5.225,149.019
C08158=1237.363,-100.940,-35.630,179.617,5.224,149.019
C08159=1237.368,-101.190,-35.619,179.615,5.225,149.020
C08160=1237.373,-101.439,-35.608,179.612,5.224,149.021
C08161=1237.378,-101.690,-35.598,179.610,5.225,149.022
C08162=1237.384,-101.939,-35.587,179.607,5.224,149.022
C08163=1237.389,-102.189,-35.576,179.605,5.224,149.023
C08164=1237.394,-102.438,-35.566,179.603,5.224,149.024
C08165=1237.399,-102.688,-35.555,179.601,5.224,149.024
C08166=1237.405,-102.937,-35.544,179.598,5.224,149.025
C08167=1237.410,-103.188,-35.534,179.596,5.224,149.026
C08168=1237.415,-103.437,-35.524,179.593,5.224,149.027
C08169=1237.420,-103.687,-35.512,179.591,5.224,149.027
C08170=1237.425,-103.936,-35.502,179.588,5.224,149.028
C08171=1237.430,-104.187,-35.492,179.586,5.224,149.029
C08172=1237.436,-104.436,-35.481,179.584,5.224,149.029
C08173=1237.441,-104.686,-35.470,179.581,5.224,149.030
C08174=1237.446,-104.935,-35.460,179.579,5.224,149.031
C08175=1237.451,-105.185,-35.449,179.577,5.224,149.032
C08176=1237.457,-105.434,-35.438,179.575,5.224,149.032
C08177=1237.462,-105.685,-35.428,179.572,5.224,149.033
C08178=1237.467,-105.934,-35.418,179.570,5.224,149.034
C08179=1237.472,-106.184,-35.406,179.568,5.223,149.034
C08180=1237.478,-106.433,-35.396,179.566,5.224,149.035
C08181=1237.483,-106.684,-35.386,179.563,5.223,149.036
C08182=1237.488,-106.933,-35.375,179.561,5.224,149.036
C08183=1237.493,-107.183,-35.364,179.559,5.224,149.037
C08184=1237.498,-107.432,-35.354,179.556,5.224,149.038
C08185=1237.503,-107.683,-35.343,179.554,5.224,149.038
C08186=1237.509,-107.932,-35.333,179.551,5.223,149.039
C08187=1237.514,-108.182,-35.323,179.549,5.224,149.040
C08188=1237.519,-108.431,-35.312,179.546,5.223,149.041
C08189=1237.524,-108.682,-35.301,179.544,5.224,149.041
C08190=1237.530,-108.931,-35.291,179.542,5.223,149.042
C08191=1237.535,-109.181,-35.280,179.540,5.224,149.043
C08192=1237.540,-109.431,-35.271,179.537,5.223,149.043
C08193=1237.545,-109.680,-35.260,179.535,5.224,149.044
C08194=1237.550,-109.930,-35.249,179.533,5.224,149.045
C08195=1237.556,-110.179,-35.239,179.530,5.223,149.046
C08196=1237.561,-110.430,-35.228,179.528,5.224,149.046
C08197=1237.566,-110.679,-35.218,179.525,5.223,149.047
C08198=1237.571,-110.929,-35.208,179.523,5.224,149.048
C08199=1237.577,-111.179,-35.197,179.520,5.223,149.048
C08200=1237.582,-111.428,-35.187,179.518,5.224,149.049
C08201=1237.587,-111.679,-35.177,179.516,5.223,149.050
C08202=1237.592,-111.927,-35.166,179.514,5.224,149.051
C08203=1237.597,-112.178,-35.156,179.511,5.223,149.051
C08204=1237.603,-112.427,-35.145,179.509,5.224,149.052
C08205=1237.608,-112.677,-35.135,179.507,5.224,149.053
C08206=1237.613,-112.927,-35.125,179.504,5.223,149.053
C08207=1237.619,-113.176,-35.114,179.502,5.223,149.054
C08208=1237.624,-113.427,-35.104,179.500,5.223,149.055
C08209=1237.629,-113.676,-35.094,179.498,5.223,149.055
C08210=1237.634,-113.925,-35.084,179.495,5.223,149.056
C08211=1237.639,-114.176,-35.073,179.493,5.223,149.057
C08212=1237.645,-114.425,-35.063,179.490,5.223,149.058
C08213=1237.650,-114.675,-35.053,179.488,5.223,149.058
C08214=1237.655,-114.925,-35.043,179.486,5.224,149.059
C08215=1237.660,-115.174,-35.033,179.483,5.223,149.060
C08216=1237.665,-115.424,-35.022,179.481,5.224,149.060
C08217=1237.671,-115.674,-35.012,179.479,5.223,149.061
C08218=1237.676,-115.924,-35.002,179.476,5.223,149.062
C08219=1237.681,-116.174,-34.992,179.474,5.223,149.063
C08220=1237.686,-116.423,-34.982,179.472,5.223,149.063
C08221=1237.691,-116.673,-34.971,179.469,5.223,149.064
C08222=1237.697,-116.923,-34.961,179.467,5.223,149.065
C08223=1237.703,-117.172,-34.951,179.465,5.224,149.065
C08224=1237.707,-117.422,-34.941,179.462,5.223,149.066
C08225=1237.712,-117.672,-34.931,179.461,5.223,149.067
C08226=1237.718,-117.921,-34.920,179.458,5.223,149.067
C08227=1237.723,-118.172,-34.910,179.456,5.223,149.068
C08228=1237.728,-118.421,-34.900,179.453,5.223,149.069
C08229=1237.733,-118.670,-34.890,179.451,5.223,149.069
C08230=1237.738,-118.921,-34.879,179.448,5.223,149.070
C08231=1237.743,-119.170,-34.870,179.446,5.223,149.071
C08232=1237.749,-119.420,-34.860,179.444,5.223,149.072
C08233=1237.754,-119.670,-34.850,179.441,5.223,149.072
C08234=1237.760,-119.920,-34.839,179.439,5.223,149.073
C08235=1237.765,-120.169,-34.830,179.437,5.223,149.074
C08236=1237.770,-120.419,-34.820,179.435,5.223,149.075
C08237=1237.775,-120.669,-34.809,179.432,5.223,149.075
C08238=1237.780,-120.918,-34.799,179.430,5.223,149.076
C08239=1237.786,-121.168,-34.789,179.427,5.223,149.077
C08240=1237.791,-121.419,-34.779,179.426,5.223,149.077
C08241=1237.796,-121.668,-34.770,179.423,5.223,149.078
C08242=1237.801,-121.917,-34.760,179.421,5.223,149.079
C08243=1237.806,-122.168,-34.749,179.419,5.223,149.079
C08244=1237.811,-122.417,-34.739,179.416,5.223,149.080
C08245=1237.817,-122.666,-34.729,179.414,5.223,149.081
C08246=1237.823,-122.916,-34.720,179.411,5.223,149.081
C08247=1237.827,-123.166,-34.710,179.409,5.223,149.082
C08248=1237.833,-123.416,-34.699,179.406,5.223,149.083
C08249=1237.838,-123.665,-34.689,179.404,5.223,149.084
C08250=1237.843,-123.915,-34.680,179.402,5.223,149.084
C08251=1237.848,-124.166,-34.670,179.400,5.223,149.085
C08252=1237.854,-124.415,-34.660,179.398,5.223,149.086
C08253=1237.859,-124.664,-34.650,179.395,5.222,149.086
C08254=1237.864,-124.914,-34.640,179.393,5.223,149.087
C08255=1237.869,-125.164,-34.630,179.390,5.222,149.088
C08256=1237.875,-125.414,-34.620,179.388,5.223,149.088
C08257=1237.880,-125.664,-34.610,179.386,5.223,149.089
C08258=1237.885,-125.913,-34.601,179.384,5.223,149.090
C08259=1237.463,-125.925,-34.636,179.379,5.226,149.092
C08260=1237.458,-125.674,-34.645,179.381,5.226,149.091
C08261=1237.453,-125.424,-34.655,179.384,5.226,149.091
C08262=1237.448,-125.175,-34.666,179.386,5.226,149.090
C08263=1237.443,-124.925,-34.674,179.389,5.226,149.089
C08264=1237.437,-124.676,-34.685,179.391,5.226,149.088
C08265=1237.432,-124.425,-34.695,179.393,5.226,149.088
C08266=1237.427,-124.176,-34.705,179.396,5.226,149.087
C08267=1237.421,-123.926,-34.714,179.398,5.226,149.086
C08268=1237.416,-123.676,-34.725,179.400,5.226,149.085
C08269=1237.411,-123.426,-34.735,179.402,5.226,149.085
C08270=1237.406,-123.177,-34.745,179.405,5.226,149.084
C08271=1237.401,-122.928,-34.754,179.407,5.226,149.084
C08272=1237.395,-122.677,-34.764,179.409,5.227,149.083
C08273=1237.390,-122.427,-34.774,179.411,5.226,149.082
C08274=1237.385,-122.178,-34.784,179.414,5.227,149.081
C08275=1237.380,-121.928,-34.794,179.416,5.226,149.081
C08276=1237.375,-121.678,-34.805,179.418,5.226,149.080
C08277=1237.369,-121.428,-34.814,179.421,5.226,149.079
C08278=1237.364,-121.179,-34.824,179.423,5.226,149.079
C08279=1237.358,-120.929,-34.834,179.426,5.226,149.078
C08280=1237.354,-120.679,-34.844,179.428,5.226,149.077
C08281=1237.348,-120.430,-34.854,179.430,5.227,149.077
C08282=1237.343,-120.180,-34.865,179.432,5.226,149.076
C08283=1237.338,-119.930,-34.875,179.435,5.227,149.075
C08284=1237.333,-119.680,-34.884,179.437,5.226,149.074
C08285=1237.327,-119.431,-34.894,179.439,5.226,149.074
C08286=1237.322,-119.180,-34.905,179.442,5.227,149.073
C08287=1237.317,-118.931,-34.914,179.444,5.226,149.072
C08288=1237.311,-118.682,-34.925,179.447,5.227,149.072
C08289=1237.306,-118.431,-34.935,179.449,5.226,149.071
C08290=1237.301,-118.182,-34.945,179.451,5.227,149.070
C08291=1237.296,-117.933,-34.955,179.453,5.226,149.069
C08292=1237.291,-117.682,-34.966,179.456,5.227,149.069
C08293=1237.285,-117.433,-34.976,179.458,5.226,149.068
C08294=1237.280,-117.183,-34.986,179.460,5.226,149.067
C08295=1237.276,-116.933,-34.996,179.462,5.227,149.067
C08296=1237.270,-116.684,-35.006,179.465,5.226,149.066
C08297=1237.264,-116.434,-35.016,179.467,5.227,149.065
C08298=1237.259,-116.184,-35.027,179.469,5.227,149.065
C08299=1237.254,-115.934,-35.036,179.472,5.227,149.064
C08300=1237.249,-115.685,-35.046,179.474,5.227,149.063
C08301=1237.244,-115.434,-35.057,179.477,5.227,149.063
C08302=1237.238,-115.185,-35.067,179.479,5.227,149.062
C08303=1237.232,-114.935,-35.077,179.481,5.226,149.061
C08304=1237.228,-114.685,-35.087,179.484,5.227,149.060
C08305=1237.223,-114.436,-35.097,179.486,5.226,149.060
C08306=1237.218,-114.186,-35.109,179.488,5.227,149.059
C08307=1237.212,-113.937,-35.119,179.491,5.226,149.058
C08308=1237.207,-113.687,-35.129,179.493,5.227,149.058
C08309=1237.202,-113.437,-35.139,179.495,5.227,149.057
C08310=1237.197,-113.188,-35.149,179.498,5.227,149.056
C08311=1237.191,-112.938,-35.159,179.500,5.227,149.055
C08312=1237.186,-112.688,-35.170,179.502,5.226,149.055
C08313=1237.181,-112.438,-35.180,179.504,5.227,149.054
C08314=1237.176,-112.188,-35.191,179.506,5.227,149.053
C08315=1237.170,-111.938,-35.201,179.509,5.227,149.053
C08316=1237.165,-111.689,-35.211,179.511,5.227,149.052
C08317=1237.160,-111.439,-35.221,179.514,5.227,149.051
C08318=1237.155,-111.189,-35.231,179.516,5.227,149.051
C08319=1237.150,-110.939,-35.242,179.519,5.227,149.050
C08320=1237.144,-110.690,-35.253,179.521,5.227,149.049
C08321=1237.139,-110.440,-35.263,179.523,5.227,149.048
C08322=1237.134,-110.190,-35.274,179.526,5.227,149.048
C08323=1237.128,-109.941,-35.284,179.528,5.227,149.047
C08324=1237.124,-109.691,-35.294,179.530,5.227,149.046
C08325=1237.118,-109.441,-35.304,179.532,5.227,149.046
C08326=1237.113,-109.191,-35.315,179.535,5.227,149.045
C08327=1237.108,-108.942,-35.325,179.537,5.227,149.044
C08328=1237.103,-108.692,-35.336,179.540,5.227,149.043
C08329=1237.097,-108.442,-35.346,179.542,5.227,149.043
C08330=1237.092,-108.192,-35.357,179.545,5.227,149.042
C08331=1237.087,-107.943,-35.367,179.547,5.227,149.041
C08332=1237.081,-107.694,-35.378,179.549,5.227,149.041
C08333=1237.076,-107.444,-35.389,179.551,5.227,149.040
C08334=1237.071,-107.194,-35.399,179.554,5.227,149.039
C08335=1237.066,-106.944,-35.409,179.556,5.227,149.038
C08336=1237.060,-106.694,-35.420,179.558,5.227,149.038
C08337=1237.056,-106.445,-35.431,179.561,5.227,149.037
C08338=1237.050,-106.195,-35.441,179.563,5.227,149.036
C08339=1237.045,-105.945,-35.452,179.566,5.227,149.036
C08340=1237.039,-105.695,-35.462,179.567,5.227,149.035
C08341=1237.035,-105.446,-35.473,179.570,5.228,149.034
C08342=1237.029,-105.196,-35.483,179.572,5.227,149.034
C08343=1237.024,-104.946,-35.494,179.575,5.228,149.033
C08344=1237.018,-104.696,-35.504,179.577,5.227,149.032
C08345=1237.014,-104.447,-35.515,179.579,5.227,149.032
C08346=1237.008,-104.197,-35.526,179.582,5.228,149.031
C08347=1237.003,-103.947,-35.536,179.584,5.227,149.030
C08348=1236.998,-103.698,-35.547,179.586,5.228,149.029
C08349=1236.993,-103.448,-35.558,179.589,5.227,149.029
C08350=1236.987,-103.198,-35.568,179.591,5.228,149.028
C08351=1236.983,-102.949,-35.579,179.593,5.227,149.027
C08352=1236.977,-102.699,-35.589,179.596,5.228,149.027
C08353=1236.972,-102.449,-35.600,179.598,5.227,149.026
C08354=1236.967,-102.199,-35.611,179.601,5.228,149.025
C08355=1236.962,-101.950,-35.621,179.603,5.228,149.024
C08356=1236.957,-101.699,-35.632,179.606,5.228,149.024
C08357=1236.951,-101.450,-35.643,179.608,5.228,149.023
C08358=1236.946,-101.200,-35.654,179.610,5.227,149.022
C08359=1236.941,-100.951,-35.664,179.612,5.228,149.022
C08360=1236.935,-100.680,-35.676,179.615,5.228,149.021
C08361=1236.930,-100.409,-35.688,179.618,5.227,149.020
C08362=1236.924,-100.138,-35.699,179.620,5.228,149.019
C08363=1236.919,-99.867,-35.710,179.622,5.228,149.018
C08364=1236.914,-99.617,-35.722,179.625,5.228,149.018
C08365=1236.908,-99.368,-35.733,179.627,5.228,149.017
C08366=1236.903,-99.118,-35.743,179.630,5.228,149.016
C08367=1236.898,-98.869,-35.754,179.632,5.228,149.016
C08368=1236.893,-98.618,-35.765,179.635,5.228,149.015
C08369=1236.888,-98.369,-35.776,179.637,5.228,149.014
C08370=1236.882,-98.119,-35.786,179.639,5.228,149.013
C08371=1236.878,-97.870,-35.797,179.642,5.228,149.013
C08372=1236.872,-97.620,-35.808,179.644,5.228,149.012
C08373=1236.867,-97.370,-35.820,179.646,5.228,149.011
C08374=1236.861,-97.121,-35.830,179.648,5.228,149.011
C08375=1236.856,-96.871,-35.841,179.651,5.228,149.010
C08376=1236.851,-96.621,-35.852,179.653,5.228,149.009
C08377=1236.846,-96.372,-35.863,179.656,5.228,149.008
C08378=1236.841,-96.122,-35.873,179.658,5.228,149.008
C08379=1236.836,-95.872,-35.885,179.661,5.228,149.007
C08380=1236.830,-95.622,-35.895,179.663,5.228,149.006
C08381=1236.825,-95.373,-35.906,179.665,5.228,149.006
C08382=1236.820,-95.123,-35.917,179.667,5.228,149.005
C08383=1236.815,-94.873,-35.928,179.670,5.229,149.004
C08384=1236.809,-94.623,-35.939,179.672,5.228,149.003
C08385=1236.804,-94.374,-35.950,179.675,5.229,149.003
C08386=1236.799,-94.124,-35.961,179.677,5.228,149.002
C08387=1236.794,-93.874,-35.972,179.680,5.229,149.001
C08388=1236.789,-93.625,-35.983,179.682,5.228,149.001
C08389=1236.783,-93.375,-35.994,179.684,5.228,149.000
C08390=1236.779,-93.125,-36.005,179.687,5.228,148.999
C08391=1236.773,-92.875,-36.016,179.689,5.228,148.998
C08392=1236.768,-92.626,-36.027,179.691,5.229,148.998
C08393=1236.762,-92.377,-36.038,179.693,5.228,148.997
C08394=1236.757,-92.126,-36.049,179.696,5.229,148.996
C08395=1236.753,-91.877,-36.060,179.698,5.228,148.996
C08396=1236.748,-91.627,-36.071,179.701,5.229,148.995
C08397=1236.742,-91.377,-36.082,179.703,5.228,148.994
C08398=1236.737,-91.128,-36.094,179.706,5.229,148.994
C08399=1236.732,-90.878,-36.105,179.708,5.229,148.993
C08400=1236.727,-90.628,-36.115,179.710,5.229,148.992
C08401=1236.721,-90.378,-36.127,179.712,5.229,148.991
C08402=1236.716,-90.129,-36.138,179.715,5.229,148.991
C08403=1236.711,-89.879,-36.148,179.717,5.229,148.990
C08404=1236.705,-89.629,-36.160,179.720,5.229,148.989
C08405=1236.701,-89.380,-36.172,179.722,5.229,148.989
C08406=1236.695,-89.130,-36.182,179.725,5.229,148.988
C08407=1236.690,-88.881,-36.193,179.727,5.229,148.987
C08408=1236.685,-88.631,-36.205,179.729,5.229,148.986
C08409=1236.680,-88.381,-36.216,179.732,5.229,148.986
C08410=1236.675,-88.131,-36.227,179.734,5.229,148.985
C08411=1236.669,-87.881,-36.238,179.736,5.229,148.984
C08412=1236.665,-87.632,-36.250,179.738,5.229,148.984
C08413=1236.659,-87.382,-36.260,179.741,5.229,148.983
C08414=1236.654,-87.132,-36.272,179.743,5.229,148.982
C08415=1236.649,-86.883,-36.283,179.746,5.229,148.981
C08416=1236.644,-86.633,-36.294,179.748,5.229,148.981
C08417=1236.638,-86.384,-36.306,179.751,5.230,148.980
C08418=1236.633,-86.134,-36.316,179.753,5.229,148.979
C08419=1236.628,-85.884,-36.328,179.755,5.230,148.979
C08420=1236.623,-85.634,-36.340,179.757,5.229,148.978
C08421=1236.618,-85.385,-36.351,179.760,5.230,148.977
C08422=1236.612,-85.135,-36.362,179.762,5.229,148.976
C08423=1236.607,-84.885,-36.373,179.765,5.230,148.976
C08424=1236.603,-84.635,-36.384,179.767,5.229,148.975
C08425=1236.597,-84.385,-36.396,179.770,5.230,148.974
C08426=1236.592,-84.136,-36.407,179.772,5.229,148.973
C08427=1236.586,-83.887,-36.419,179.775,5.230,148.973
C08428=1236.582,-83.637,-36.430,179.777,5.229,148.972
C08429=1236.577,-83.387,-36.442,179.780,5.230,148.971
C08430=1236.571,-83.137,-36.452,179.782,5.229,148.971
C08431=1236.566,-82.888,-36.464,179.784,5.230,148.970
C08432=1236.561,-82.638,-36.476,179.787,5.230,148.969
C08433=1236.556,-82.388,-36.487,179.789,5.230,148.968
C08434=1236.551,-82.138,-36.499,179.791,5.230,148.968
C08435=1236.546,-81.889,-36.510,179.794,5.230,148.967
C08436=1236.541,-81.640,-36.521,179.796,5.230,148.966
C08437=1236.535,-81.390,-36.533,179.799,5.230,148.966
C08438=1236.530,-81.140,-36.544,179.801,5.230,148.965
C08439=1236.525,-80.890,-36.556,179.804,5.230,148.964
C08440=1236.520,-80.641,-36.567,179.806,5.230,148.963
C08441=1236.514,-80.391,-36.578,179.808,5.231,148.963
C08442=1236.509,-80.141,-36.589,179.810,5.230,148.962
C08443=1236.504,-79.891,-36.601,179.813,5.231,148.961
C08444=1236.499,-79.642,-36.613,179.815,5.230,148.961
C08445=1236.494,-79.392,-36.624,179.818,5.231,148.960
C08446=1236.489,-79.142,-36.636,179.820,5.230,148.959
C08447=1236.483,-78.893,-36.647,179.823,5.231,148.958
C08448=1236.478,-78.643,-36.659,179.825,5.231,148.958
C08449=1236.473,-78.393,-36.670,179.827,5.231,148.957
C08450=1236.468,-78.144,-36.682,179.829,5.231,148.956
C08451=1236.463,-77.894,-36.694,179.832,5.231,148.956
C08452=1236.458,-77.644,-36.705,179.834,5.231,148.955
C08453=1236.453,-77.394,-36.717,179.837,5.231,148.954
C08454=1236.447,-77.145,-36.728,179.839,5.231,148.953
C08455=1236.442,-76.895,-36.740,179.841,5.231,148.953
C08456=1236.437,-76.646,-36.752,179.844,5.231,148.952
C08457=1236.432,-76.396,-36.763,179.846,5.230,148.951
C08458=1236.427,-76.146,-36.775,179.849,5.231,148.950
C08459=1236.422,-75.897,-36.787,179.851,5.231,148.950
C08460=1236.417,-75.647,-36.799,179.854,5.231,148.949
C08461=1236.411,-75.397,-36.810,179.856,5.231,148.948
C08462=1236.406,-75.148,-36.821,179.858,5.231,148.948
C08463=1236.400,-74.898,-36.833,179.861,5.232,148.947
C08464=1236.395,-74.628,-36.846,179.863,5.231,148.946
C08465=1236.390,-74.357,-36.859,179.866,5.232,148.945
C08466=1236.384,-74.087,-36.871,179.869,5.231,148.945
C08467=1236.378,-73.817,-36.884,179.871,5.231,148.944
C08468=1236.374,-73.567,-36.895,179.874,5.232,148.943
C08469=1236.368,-73.317,-36.907,179.876,5.232,148.942
C08470=1236.363,-73.068,-36.920,179.879,5.232,148.942
C08471=1236.358,-72.818,-36.931,179.881,5.232,148.941
C08472=1236.352,-72.569,-36.943,179.883,5.232,148.940
C08473=1236.348,-72.319,-36.954,179.885,5.232,148.940
C08474=1236.342,-72.069,-36.966,179.888,5.232,148.939
C08475=1236.337,-71.819,-36.978,179.890,5.232,148.938
C08476=1236.332,-71.570,-36.990,179.893,5.232,148.937
C08477=1236.327,-71.321,-37.002,179.895,5.232,148.937
C08478=1236.321,-71.071,-37.013,179.898,5.233,148.936
C08479=1236.317,-70.821,-37.025,179.900,5.232,148.935
C08480=1236.312,-70.572,-37.037,179.903,5.232,148.934
C08481=1236.306,-70.322,-37.049,179.905,5.232,148.934
C08482=1236.301,-70.072,-37.061,179.908,5.233,148.933
C08483=1236.296,-69.822,-37.072,179.910,5.232,148.932
C08484=1236.291,-69.572,-37.084,179.912,5.233,148.932
C08485=1236.286,-69.323,-37.097,179.915,5.232,148.931
C08486=1236.281,-69.073,-37.108,179.917,5.233,148.930
C08487=1236.275,-68.823,-37.120,179.919,5.232,148.929
C08488=1236.270,-68.574,-37.133,179.922,5.233,148.929
C08489=1236.265,-68.324,-37.145,179.924,5.233,148.928
C08490=1236.260,-68.074,-37.156,179.927,5.233,148.927
C08491=1236.255,-67.824,-37.168,179.929,5.233,148.927
C08492=1236.250,-67.575,-37.180,179.931,5.233,148.926
C08493=1236.245,-67.326,-37.192,179.934,5.233,148.925
C08494=1236.240,-67.076,-37.204,179.936,5.233,148.924
C08495=1236.234,-66.826,-37.216,179.938,5.233,148.924
C08496=1236.229,-66.576,-37.228,179.941,5.234,148.923
C08497=1236.224,-66.327,-37.239,179.943,5.233,148.922
C08498=1236.219,-66.077,-37.252,179.946,5.234,148.922
C08499=1236.214,-65.827,-37.264,179.948,5.233,148.921
C08500=1236.208,-65.578,-37.276,179.951,5.233,148.920
C08501=1236.203,-65.328,-37.288,179.953,5.233,148.919
C08502=1236.198,-65.079,-37.300,179.956,5.234,148.919
C08503=1236.193,-64.829,-37.312,179.958,5.233,148.918
C08504=1236.188,-64.579,-37.324,179.961,5.234,148.917
C08505=1236.183,-64.329,-37.336,179.963,5.234,148.916
C08506=1236.177,-64.080,-37.349,179.965,5.234,148.916
C08507=1236.173,-63.830,-37.360,179.968,5.234,148.915
C08508=1236.168,-63.581,-37.372,179.970,5.234,148.914
C08509=1236.162,-63.331,-37.384,179.973,5.235,148.914
C08510=1236.157,-63.081,-37.396,179.975,5.234,148.913
C08511=1236.152,-62.832,-37.409,179.977,5.235,148.912
C08512=1236.146,-62.582,-37.421,179.980,5.234,148.912
C08513=1236.142,-62.333,-37.433,179.982,5.235,148.911
C08514=1236.136,-62.083,-37.445,179.984,5.234,148.910
C08515=1236.131,-61.834,-37.457,179.987,5.235,148.909
C08516=1236.126,-61.583,-37.469,179.989,5.235,148.909
C08517=1236.121,-61.334,-37.482,179.992,5.235,148.908
C08518=1236.116,-61.084,-37.494,179.994,5.234,148.907
C08519=1236.111,-60.835,-37.506,179.997,5.235,148.906
C08520=1236.106,-60.585,-37.518,179.999,5.235,148.906
C08521=1236.101,-60.336,-37.530,-179.998,5.235,148.905
C08522=1236.095,-60.086,-37.542,-179.996,5.235,148.904
C08523=1236.090,-59.836,-37.555,-179.993,5.235,148.904
C08524=1236.085,-59.586,-37.567,-179.991,5.236,148.903
C08525=1236.080,-59.337,-37.579,-179.989,5.235,148.902
C08526=1236.075,-59.086,-37.592,-179.986,5.236,148.901
C08527=1236.070,-58.837,-37.604,-179.984,5.236,148.901
C08528=1236.065,-58.588,-37.617,-179.981,5.236,148.900
C08529=1236.060,-58.338,-37.628,-179.979,5.236,148.899
C08530=1236.055,-58.089,-37.641,-179.977,5.236,148.899
C08531=1236.049,-57.839,-37.653,-179.974,5.236,148.898
C08532=1236.044,-57.590,-37.665,-179.972,5.236,148.897
C08533=1236.039,-57.340,-37.677,-179.969,5.236,148.896
C08534=1236.034,-57.090,-37.690,-179.967,5.236,148.896
C08535=1236.029,-56.840,-37.703,-179.964,5.236,148.895
C08536=1236.024,-56.590,-37.715,-179.962,5.236,148.894
C08537=1236.019,-56.341,-37.727,-179.960,5.236,148.893
C08538=1236.014,-56.092,-37.740,-179.957,5.236,148.893
C08539=1236.008,-55.842,-37.752,-179.954,5.237,148.892
C08540=1236.003,-55.593,-37.764,-179.952,5.237,148.891
C08541=1235.999,-55.343,-37.777,-179.950,5.237,148.891
C08542=1235.993,-55.093,-37.789,-179.948,5.237,148.890
C08543=1235.988,-54.843,-37.802,-179.945,5.237,148.889
C08544=1235.983,-54.594,-37.814,-179.943,5.237,148.889
C08545=1235.977,-54.344,-37.826,-179.940,5.237,148.888
C08546=1235.973,-54.094,-37.839,-179.938,5.237,148.887
C08547=1235.968,-53.845,-37.852,-179.935,5.238,148.886
C08548=1235.962,-53.595,-37.864,-179.933,5.237,148.886
C08549=1235.957,-53.345,-37.876,-179.930,5.237,148.885
C08550=1235.952,-53.096,-37.889,-179.927,5.238,148.884
C08551=1235.947,-52.846,-37.901,-179.925,5.238,148.883
C08552=1235.942,-52.596,-37.914,-179.923,5.238,148.883
C08553=1235.937,-52.347,-37.926,-179.921,5.238,148.882
C08554=1235.932,-52.098,-37.939,-179.918,5.238,148.881
C08555=1235.926,-51.848,-37.951,-179.916,5.238,148.881
C08556=1235.922,-51.598,-37.964,-179.913,5.238,148.880
C08557=1235.917,-51.348,-37.976,-179.911,5.238,148.879
C08558=1235.912,-51.099,-37.989,-179.908,5.239,148.878
C08559=1235.907,-50.850,-38.002,-179.906,5.238,148.878
C08560=1235.901,-50.600,-38.013,-179.904,5.239,148.877
C08561=1235.896,-50.349,-38.027,-179.901,5.239,148.876
C08562=1235.891,-50.100,-38.040,-179.899,5.239,148.876
C08563=1235.886,-49.851,-38.052,-179.896,5.239,148.875
C08564=1235.880,-49.601,-38.065,-179.894,5.239,148.874
C08565=1235.876,-49.351,-38.077,-179.891,5.239,148.873
C08566=1235.871,-49.101,-38.090,-179.889,5.239,148.873
C08567=1235.865,-48.852,-38.102,-179.886,5.239,148.872
C08568=1235.860,-48.582,-38.116,-179.884,5.240,148.871
C08569=1235.854,-48.313,-38.130,-179.881,5.239,148.870
C08570=1235.849,-48.043,-38.143,-179.878,5.240,148.870
C08571=1235.843,-47.773,-38.158,-179.876,5.240,148.869
C08572=1235.838,-47.523,-38.170,-179.874,5.240,148.868
C08573=1235.833,-47.274,-38.182,-179.871,5.240,148.867
C08574=1235.828,-47.024,-38.195,-179.869,5.240,148.867
C08575=1235.823,-46.775,-38.208,-179.866,5.240,148.866
C08576=1235.817,-46.525,-38.221,-179.864,5.240,148.865
C08577=1235.812,-46.276,-38.234,-179.861,5.241,148.865
C08578=1235.808,-46.026,-38.247,-179.859,5.241,148.864
C08579=1235.803,-45.776,-38.259,-179.856,5.240,148.863
C08580=1235.797,-45.527,-38.272,-179.853,5.241,148.862
C08581=1235.793,-45.277,-38.285,-179.851,5.241,148.862
C08582=1235.787,-45.027,-38.298,-179.849,5.241,148.861
C08583=1235.782,-44.778,-38.311,-179.847,5.241,148.860
C08584=1235.777,-44.529,-38.323,-179.844,5.241,148.859
C08585=1235.772,-44.279,-38.336,-179.841,5.242,148.859
C08586=1235.766,-44.029,-38.349,-179.839,5.241,148.858
C08587=1235.761,-43.780,-38.362,-179.837,5.242,148.857
C08588=1235.757,-43.530,-38.375,-179.834,5.242,148.857
C08589=1235.752,-43.280,-38.387,-179.832,5.242,148.856
C08590=1235.746,-43.031,-38.400,-179.830,5.242,148.855
C08591=1235.741,-42.781,-38.414,-179.827,5.242,148.855
C08592=1235.736,-42.532,-38.426,-179.824,5.243,148.854
C08593=1235.731,-42.282,-38.439,-179.822,5.242,148.853
C08594=1235.726,-42.032,-38.452,-179.819,5.243,148.852
C08595=1235.721,-41.783,-38.465,-179.817,5.242,148.852
C08596=1235.715,-41.533,-38.478,-179.814,5.243,148.851
C08597=1235.711,-41.283,-38.491,-179.812,5.242,148.850
C08598=1235.705,-41.034,-38.504,-179.810,5.243,148.849
C08599=1235.701,-40.784,-38.517,-179.807,5.243,148.849
C08600=1235.695,-40.534,-38.529,-179.805,5.243,148.848
C08601=1235.690,-40.285,-38.542,-179.802,5.244,148.847
C08602=1235.685,-40.035,-38.555,-179.800,5.243,148.847
C08603=1235.680,-39.785,-38.568,-179.798,5.244,148.846
C08604=1235.675,-39.536,-38.581,-179.795,5.244,148.845
C08605=1235.670,-39.286,-38.595,-179.793,5.244,148.845
C08606=1235.665,-39.037,-38.608,-179.790,5.245,148.844
C08607=1235.660,-38.787,-38.621,-179.788,5.244,148.843
C08608=1235.654,-38.537,-38.634,-179.785,5.244,148.842
C08609=1235.649,-38.288,-38.646,-179.783,5.244,148.841
C08610=1235.645,-38.038,-38.659,-179.780,5.245,148.841
C08611=1235.639,-37.788,-38.672,-179.778,5.244,148.840
C08612=1235.634,-37.540,-38.686,-179.775,5.245,148.839
C08613=1235.629,-37.290,-38.699,-179.773,5.245,148.839
C08614=1235.624,-37.040,-38.712,-179.771,5.245,148.838
C08615=1235.619,-36.790,-38.725,-179.768,5.245,148.837
C08616=1235.613,-36.540,-38.738,-179.766,5.245,148.837
C08617=1235.609,-36.291,-38.752,-179.763,5.246,148.836
C08618=1235.604,-36.042,-38.764,-179.761,5.246,148.835
C08619=1235.598,-35.792,-38.778,-179.758,5.246,148.834
C08620=1235.594,-35.542,-38.791,-179.756,5.246,148.834
C08621=1235.588,-35.292,-38.804,-179.754,5.246,148.833
C08622=1235.583,-35.043,-38.817,-179.751,5.247,148.832
C08623=1235.578,-34.794,-38.830,-179.748,5.247,148.831
C08624=1235.573,-34.543,-38.844,-179.746,5.246,148.831
C08625=1235.568,-34.294,-38.856,-179.743,5.247,148.830
C08626=1235.562,-34.045,-38.870,-179.741,5.247,148.829
C08627=1235.558,-33.795,-38.883,-179.738,5.247,148.829
C08628=1235.553,-33.546,-38.896,-179.736,5.247,148.828
C08629=1235.548,-33.296,-38.910,-179.734,5.247,148.827
C08630=1235.543,-33.047,-38.923,-179.731,5.248,148.827
C08631=1235.537,-32.796,-38.936,-179.729,5.247,148.826
C08632=1235.533,-32.548,-38.949,-179.726,5.248,148.825
C08633=1235.527,-32.297,-38.963,-179.724,5.248,148.824
C08634=1235.522,-32.048,-38.976,-179.721,5.248,148.824
C08635=1235.517,-31.798,-38.990,-179.719,5.249,148.823
C08636=1235.512,-31.549,-39.002,-179.717,5.248,148.822
C08637=1235.507,-31.299,-39.016,-179.714,5.248,148.821
C08638=1235.502,-31.050,-39.029,-179.712,5.248,148.821
C08639=1235.497,-30.800,-39.043,-179.709,5.249,148.820
C08640=1235.492,-30.550,-39.056,-179.706,5.249,148.819
C08641=1235.487,-30.301,-39.070,-179.704,5.249,148.819
C08642=1235.482,-30.051,-39.082,-179.701,5.249,148.818
C08643=1235.477,-29.801,-39.097,-179.699,5.249,148.817
C08644=1235.471,-29.552,-39.109,-179.697,5.250,148.817
C08645=1235.466,-29.302,-39.123,-179.694,5.250,148.816
C08646=1235.461,-29.053,-39.136,-179.692,5.250,148.815
C08647=1235.456,-28.803,-39.150,-179.689,5.250,148.814
C08648=1235.451,-28.554,-39.163,-179.687,5.251,148.814
C08649=1235.446,-28.304,-39.177,-179.685,5.251,148.813
C08650=1235.441,-28.055,-39.190,-179.682,5.251,148.812
C08651=1235.436,-27.805,-39.203,-179.680,5.251,148.812
C08652=1235.430,-27.555,-39.217,-179.677,5.251,148.811
C08653=1235.426,-27.306,-39.230,-179.674,5.251,148.810
C08654=1235.421,-27.055,-39.244,-179.672,5.251,148.809
C08655=1235.416,-26.807,-39.257,-179.669,5.252,148.809
C08656=1235.411,-26.556,-39.271,-179.667,5.251,148.808
C08657=1235.406,-26.308,-39.284,-179.664,5.252,148.807
C08658=1235.400,-26.057,-39.298,-179.662,5.252,148.807
C08659=1235.395,-25.808,-39.312,-179.660,5.252,148.806
C08660=1235.390,-25.558,-39.325,-179.657,5.252,148.805
C08661=1235.385,-25.309,-39.338,-179.655,5.252,148.804
C08662=1235.380,-25.059,-39.351,-179.652,5.253,148.804
C08663=1235.375,-24.810,-39.366,-179.650,5.253,148.803
C08664=1235.370,-24.561,-39.380,-179.648,5.253,148.802
C08665=1235.365,-24.311,-39.393,-179.645,5.253,148.802
C08666=1235.360,-24.062,-39.407,-179.642,5.254,148.801
C08667=1235.354,-23.811,-39.420,-179.640,5.254,148.800
C08668=1235.350,-23.562,-39.434,-179.637,5.254,148.799
C08669=1235.344,-23.312,-39.447,-179.635,5.253,148.799
C08670=1235.339,-23.062,-39.461,-179.632,5.254,148.798
C08671=1235.335,-22.814,-39.475,-179.630,5.255,148.797
C08672=1235.329,-22.544,-39.490,-179.628,5.254,148.797
C08673=1235.324,-22.275,-39.505,-179.625,5.255,148.796
C08674=1235.318,-22.005,-39.519,-179.622,5.255,148.795
C08675=1235.313,-21.735,-39.534,-179.619,5.255,148.794
C08676=1235.308,-21.487,-39.547,-179.617,5.255,148.794
C08677=1235.303,-21.237,-39.561,-179.614,5.256,148.793
C08678=1235.297,-20.987,-39.575,-179.612,5.256,148.792
C08679=1235.293,-20.738,-39.588,-179.610,5.256,148.791
C08680=1235.288,-20.488,-39.603,-179.607,5.256,148.791
C08681=1235.282,-20.239,-39.616,-179.605,5.256,148.790
C08682=1235.277,-19.989,-39.630,-179.602,5.257,148.789
C08683=1235.273,-19.740,-39.644,-179.600,5.257,148.789
C08684=1235.267,-19.490,-39.657,-179.597,5.256,148.788
C08685=1235.262,-19.240,-39.671,-179.594,5.257,148.787
C08686=1235.258,-18.991,-39.685,-179.592,5.257,148.786
C08687=1235.252,-18.742,-39.699,-179.590,5.257,148.786
C08688=1235.247,-18.492,-39.712,-179.587,5.258,148.785
C08689=1235.242,-18.242,-39.727,-179.584,5.258,148.784
C08690=1235.236,-17.993,-39.741,-179.582,5.258,148.784
C08691=1235.232,-17.743,-39.754,-179.580,5.258,148.783
C08692=1235.227,-17.493,-39.768,-179.577,5.258,148.782
C08693=1235.221,-17.244,-39.782,-179.575,5.259,148.782
C08694=1235.216,-16.994,-39.796,-179.572,5.259,148.781
C08695=1235.212,-16.745,-39.810,-179.570,5.259,148.780
C08696=1235.207,-16.496,-39.824,-179.567,5.259,148.779
C08697=1235.201,-16.246,-39.837,-179.565,5.260,148.779
C08698=1235.196,-15.996,-39.851,-179.563,5.260,148.778
C08699=1235.191,-15.747,-39.865,-179.560,5.260,148.777
C08700=1235.186,-15.497,-39.880,-179.557,5.261,148.777
C08701=1235.182,-15.248,-39.893,-179.555,5.260,148.776
C08702=1235.176,-14.997,-39.907,-179.552,5.260,148.775
C08703=1235.171,-14.748,-39.921,-179.549,5.261,148.774
C08704=1235.166,-14.499,-39.935,-179.547,5.261,148.774
C08705=1235.161,-14.249,-39.949,-179.545,5.261,148.773
C08706=1235.155,-14.000,-39.963,-179.543,5.261,148.772
C08707=1235.151,-13.751,-39.977,-179.540,5.261,148.772
C08708=1235.146,-13.501,-39.991,-179.537,5.262,148.771
C08709=1235.141,-13.251,-40.005,-179.535,5.262,148.770
C08710=1235.135,-13.002,-40.019,-179.533,5.262,148.769
C08711=1235.130,-12.752,-40.033,-179.530,5.263,148.769
C08712=1235.126,-12.502,-40.047,-179.528,5.262,148.768
C08713=1235.121,-12.252,-40.061,-179.525,5.263,148.767
C08714=1235.115,-12.003,-40.075,-179.523,5.263,148.767
C08715=1235.111,-11.754,-40.089,-179.520,5.263,148.766
C08716=1235.106,-11.504,-40.103,-179.518,5.264,148.765
C08717=1235.101,-11.255,-40.118,-179.515,5.264,148.765
C08718=1235.096,-11.005,-40.132,-179.513,5.264,148.764
C08719=1235.090,-10.756,-40.146,-179.510,5.264,148.763
C08720=1235.085,-10.506,-40.160,-179.507,5.265,148.762
C08721=1235.080,-10.256,-40.174,-179.505,5.264,148.762
C08722=1235.075,-10.007,-40.189,-179.502,5.265,148.761
C08723=1235.070,-9.758,-40.203,-179.500,5.265,148.760
C08724=1235.065,-9.508,-40.217,-179.498,5.265,148.760
C08725=1235.060,-9.258,-40.231,-179.495,5.266,148.759
C08726=1235.055,-9.009,-40.245,-179.492,5.266,148.758
C08727=1235.050,-8.759,-40.260,-179.490,5.266,148.757
C08728=1235.045,-8.510,-40.274,-179.488,5.266,148.757
C08729=1235.040,-8.260,-40.288,-179.485,5.267,148.756
C08730=1235.035,-8.010,-40.302,-179.483,5.267,148.755
C08731=1235.030,-7.761,-40.316,-179.480,5.267,148.755
C08732=1235.025,-7.511,-40.331,-179.478,5.268,148.754
C08733=1235.020,-7.261,-40.345,-179.476,5.267,148.753
C08734=1235.015,-7.013,-40.358,-179.473,5.268,148.753
C08735=1235.010,-6.763,-40.373,-179.470,5.268,148.752
C08736=1235.004,-6.513,-40.387,-179.468,5.268,148.751
C08737=1235.000,-6.264,-40.402,-179.466,5.269,148.751
C08738=1234.995,-6.014,-40.417,-179.463,5.269,148.750
C08739=1234.990,-5.764,-40.431,-179.460,5.269,148.749
C08740=1234.984,-5.515,-40.445,-179.458,5.269,148.748
C08741=1234.979,-5.266,-40.459,-179.455,5.270,148.748
C08742=1234.974,-5.016,-40.473,-179.453,5.269,148.747
C08743=1234.969,-4.766,-40.488,-179.450,5.270,148.746
C08744=1234.965,-4.517,-40.503,-179.448,5.270,148.745
C08745=1234.960,-4.267,-40.517,-179.446,5.270,148.745
C08746=1234.955,-4.018,-40.531,-179.443,5.271,148.744
C08747=1234.950,-3.768,-40.546,-179.440,5.271,148.743
C08748=1234.944,-3.519,-40.559,-179.438,5.272,148.743
C08749=1234.939,-3.269,-40.574,-179.435,5.271,148.742
C08750=1234.935,-3.020,-40.589,-179.433,5.272,148.741
C08751=1234.930,-2.771,-40.603,-179.430,5.272,148.741
C08752=1234.925,-2.521,-40.617,-179.428,5.272,148.740
C08753=1234.919,-2.271,-40.632,-179.425,5.273,148.739
C08754=1234.914,-2.022,-40.647,-179.423,5.273,148.739
C08755=1234.909,-1.772,-40.661,-179.421,5.273,148.738
C08756=1234.905,-1.522,-40.676,-179.418,5.273,148.737
C08757=1234.899,-1.273,-40.690,-179.415,5.274,148.737
C08758=1234.894,-1.024,-40.705,-179.413,5.274,148.736
C08759=1234.889,-0.774,-40.719,-179.411,5.274,148.735
C08760=1234.884,-0.525,-40.733,-179.408,5.275,148.734
C08761=1234.879,-0.275,-40.748,-179.406,5.275,148.734
C08762=1234.874,-0.026,-40.763,-179.403,5.275,148.733
C08763=1234.869,0.224,-40.777,-179.400,5.275,148.732
C08764=1234.864,0.474,-40.792,-179.397,5.276,148.731
C08765=1234.859,0.723,-40.807,-179.395,5.275,148.731
C08766=1234.855,0.973,-40.821,-179.393,5.276,148.730
C08767=1234.849,1.223,-40.836,-179.390,5.277,148.729
C08768=1234.844,1.472,-40.851,-179.388,5.276,148.729
C08769=1234.839,1.721,-40.865,-179.385,5.277,148.728
C08770=1234.834,1.971,-40.879,-179.383,5.277,148.727
C08771=1234.830,2.220,-40.894,-179.381,5.277,148.727
C08772=1234.824,2.470,-40.909,-179.378,5.278,148.726
C08773=1234.819,2.720,-40.923,-179.375,5.278,148.725
C08774=1234.814,2.968,-40.938,-179.373,5.279,148.725
C08775=1234.809,3.218,-40.952,-179.371,5.278,148.724
C08776=1234.803,3.487,-40.969,-179.368,5.279,148.723
C08777=1234.798,3.756,-40.984,-179.365,5.279,148.723
C08778=1234.793,4.025,-41.000,-179.362,5.280,148.722
C08779=1234.788,4.294,-41.016,-179.360,5.280,148.721
C08780=1234.782,4.543,-41.031,-179.357,5.280,148.720
C08781=1234.777,4.793,-41.046,-179.355,5.280,148.720
C08782=1234.772,5.042,-41.060,-179.352,5.281,148.719
C08783=1234.767,5.292,-41.075,-179.350,5.281,148.718
C08784=1234.762,5.541,-41.090,-179.347,5.281,148.717
C08785=1234.757,5.791,-41.105,-179.345,5.282,148.717
C08786=1234.752,6.040,-41.119,-179.342,5.282,148.716
C08787=1234.747,6.290,-41.135,-179.340,5.282,148.715
C08788=1234.742,6.539,-41.149,-179.337,5.283,148.715
C08789=1234.737,6.788,-41.164,-179.335,5.283,148.714
C08790=1234.732,7.038,-41.179,-179.333,5.283,148.713
C08791=1234.727,7.288,-41.194,-179.330,5.283,148.713
C08792=1234.722,7.537,-41.208,-179.327,5.284,148.712
C08793=1234.717,7.787,-41.224,-179.325,5.284,148.711
C08794=1234.712,8.037,-41.238,-179.323,5.284,148.711
C08795=1234.708,8.286,-41.253,-179.320,5.285,148.710
C08796=1234.702,8.536,-41.269,-179.317,5.285,148.709
C08797=1234.697,8.785,-41.283,-179.314,5.285,148.708
C08798=1234.693,9.034,-41.298,-179.312,5.285,148.708
C08799=1234.687,9.284,-41.313,-179.309,5.286,148.707
C08800=1234.682,9.533,-41.328,-179.307,5.286,148.706
C08801=1234.677,9.783,-41.342,-179.305,5.286,148.706
C08802=1234.672,10.033,-41.358,-179.302,5.286,148.705
C08803=1234.667,10.282,-41.373,-179.299,5.287,148.704
C08804=1234.662,10.531,-41.387,-179.297,5.288,148.703
C08805=1234.657,10.781,-41.403,-179.295,5.287,148.703
C08806=1234.652,11.030,-41.418,-179.292,5.288,148.702
C08807=1234.647,11.280,-41.433,-179.289,5.288,148.701
C08808=1234.643,11.530,-41.448,-179.287,5.289,148.701
C08809=1234.638,11.779,-41.463,-179.285,5.289,148.700
C08810=1234.632,12.029,-41.478,-179.282,5.289,148.699
C08811=1234.628,12.278,-41.493,-179.279,5.290,148.699
C08812=1234.622,12.527,-41.508,-179.277,5.290,148.698
C08813=1234.617,12.777,-41.523,-179.275,5.290,148.697
C08814=1234.612,13.026,-41.538,-179.272,5.291,148.697
C08815=1234.607,13.276,-41.553,-179.269,5.291,148.696
C08816=1234.602,13.525,-41.567,-179.267,5.291,148.695
C08817=1234.597,13.775,-41.583,-179.265,5.291,148.695
C08818=1234.593,14.024,-41.598,-179.262,5.292,148.694
C08819=1234.587,14.274,-41.614,-179.259,5.292,148.693
C08820=1234.582,14.524,-41.628,-179.257,5.292,148.693
C08821=1234.577,14.773,-41.644,-179.255,5.293,148.692
C08822=1234.572,15.022,-41.659,-179.252,5.293,148.691
C08823=1234.567,15.271,-41.674,-179.249,5.294,148.690
C08824=1234.562,15.521,-41.689,-179.247,5.294,148.690
C08825=1234.557,15.771,-41.705,-179.245,5.294,148.689
C08826=1234.553,16.020,-41.720,-179.242,5.295,148.688
C08827=1234.547,16.270,-41.735,-179.239,5.295,148.688
C08828=1234.543,16.519,-41.750,-179.237,5.295,148.687
C08829=1234.537,16.769,-41.765,-179.235,5.295,148.686
C08830=1234.532,17.018,-41.780,-179.232,5.296,148.686
C08831=1234.527,17.268,-41.796,-179.229,5.297,148.685
C08832=1234.523,17.517,-41.811,-179.227,5.296,148.684
C08833=1234.517,17.767,-41.827,-179.225,5.297,148.684
C08834=1234.512,18.016,-41.842,-179.222,5.297,148.683
C08835=1234.507,18.266,-41.857,-179.219,5.298,148.682
C08836=1234.502,18.516,-41.872,-179.217,5.298,148.682
C08837=1234.498,18.765,-41.887,-179.215,5.298,148.681
C08838=1234.492,19.014,-41.903,-179.212,5.299,148.680
C08839=1234.488,19.263,-41.918,-179.209,5.299,148.680
C08840=1234.482,19.513,-41.934,-179.207,5.300,148.679
C08841=1234.477,19.763,-41.950,-179.205,5.300,148.678
C08842=1234.473,20.012,-41.965,-179.202,5.300,148.677
C08843=1234.467,20.261,-41.980,-179.199,5.301,148.677
C08844=1234.463,20.510,-41.995,-179.197,5.301,148.676
C08845=1234.457,20.760,-42.010,-179.194,5.301,148.675
C08846=1234.452,21.011,-42.026,-179.192,5.302,148.675
C08847=1234.448,21.260,-42.041,-179.189,5.302,148.674
C08848=1234.442,21.509,-42.057,-179.187,5.303,148.673
C08849=1234.438,21.758,-42.072,-179.184,5.302,148.673
C08850=1234.433,22.008,-42.088,-179.182,5.303,148.672
C08851=1234.427,22.258,-42.103,-179.179,5.303,148.671
C08852=1234.423,22.507,-42.118,-179.177,5.304,148.671
C08853=1234.417,22.756,-42.134,-179.174,5.305,148.670
C08854=1234.413,23.006,-42.150,-179.172,5.304,148.669
C08855=1234.408,23.255,-42.165,-179.169,5.305,148.669
C08856=1234.403,23.505,-42.180,-179.167,5.305,148.668
C08857=1234.397,23.754,-42.196,-179.164,5.306,148.667
C08858=1234.393,24.004,-42.211,-179.162,5.306,148.667
C08859=1234.388,24.253,-42.227,-179.159,5.306,148.666
C08860=1234.383,24.502,-42.243,-179.157,5.307,148.665
C08861=1234.379,24.752,-42.258,-179.154,5.307,148.665
C08862=1234.373,25.001,-42.274,-179.151,5.308,148.664
C08863=1234.368,25.251,-42.290,-179.149,5.308,148.663
C08864=1234.362,25.500,-42.305,-179.147,5.308,148.662
C08865=1234.358,25.750,-42.321,-179.144,5.309,148.662
C08866=1234.353,25.999,-42.336,-179.141,5.309,148.661
C08867=1234.348,26.249,-42.352,-179.139,5.310,148.660
C08868=1234.344,26.499,-42.367,-179.136,5.310,148.660
C08869=1234.338,26.748,-42.383,-179.134,5.310,148.659
C08870=1234.333,26.997,-42.399,-179.131,5.311,148.658
C08871=1234.328,27.247,-42.415,-179.129,5.311,148.658
C08872=1234.323,27.496,-42.430,-179.126,5.312,148.657
C08873=1234.318,27.745,-42.445,-179.124,5.312,148.656
C08874=1234.314,27.995,-42.461,-179.121,5.312,148.656
C08875=1234.308,28.245,-42.477,-179.119,5.313,148.655
C08876=1234.303,28.494,-42.493,-179.116,5.313,148.654
C08877=1234.299,28.743,-42.509,-179.113,5.314,148.654
C08878=1234.294,28.993,-42.524,-179.111,5.314,148.653
C08879=1234.288,29.242,-42.540,-179.109,5.314,148.652
C08880=1234.283,29.511,-42.557,-179.106,5.315,148.652
C08881=1234.278,29.780,-42.574,-179.103,5.315,148.651
C08882=1234.272,30.048,-42.591,-179.101,5.316,148.650
C08883=1234.267,30.316,-42.608,-179.098,5.316,148.650
C08884=1234.263,30.567,-42.624,-179.095,5.317,148.649
C08885=1234.257,30.815,-42.640,-179.093,5.317,148.648
C08886=1234.252,31.065,-42.656,-179.091,5.317,148.648
C08887=1234.247,31.315,-42.672,-179.088,5.318,148.647
C08888=1234.242,31.564,-42.687,-179.085,5.318,148.646
C08889=1234.237,31.813,-42.703,-179.083,5.319,148.646
C08890=1234.233,32.063,-42.719,-179.080,5.319,148.645
C08891=1234.227,32.312,-42.734,-179.078,5.319,148.644
C08892=1234.223,32.562,-42.751,-179.075,5.320,148.643
C08893=1234.218,32.811,-42.767,-179.073,5.320,148.643
C08894=1234.212,33.061,-42.782,-179.070,5.321,148.642
C08895=1234.208,33.310,-42.799,-179.067,5.321,148.641
C08896=1234.202,33.559,-42.814,-179.065,5.321,148.641
C08897=1234.198,33.810,-42.830,-179.063,5.322,148.640
C08898=1234.193,34.058,-42.846,-179.060,5.322,148.639
C08899=1234.188,34.307,-42.862,-179.057,5.323,148.639
C08900=1234.183,34.557,-42.878,-179.055,5.323,148.638
C08901=1234.178,34.806,-42.894,-179.052,5.324,148.637
C08902=1234.173,35.056,-42.910,-179.050,5.324,148.637
C08903=1234.168,35.305,-42.926,-179.047,5.324,148.636
C08904=1234.163,35.555,-42.942,-179.045,5.325,148.635
C08905=1234.158,35.804,-42.958,-179.042,5.325,148.635
C08906=1234.153,36.054,-42.974,-179.039,5.326,148.634
C08907=1234.148,36.304,-42.990,-179.037,5.327,148.633
C08908=1234.143,36.552,-43.006,-179.035,5.327,148.633
C08909=1234.138,36.802,-43.022,-179.033,5.327,148.632
C08910=1234.133,37.051,-43.039,-179.030,5.328,148.632
C08911=1234.128,37.301,-43.055,-179.027,5.328,148.631
C08912=1234.123,37.550,-43.071,-179.025,5.329,148.630
C08913=1234.118,37.800,-43.087,-179.022,5.329,148.630
C08914=1234.113,38.049,-43.103,-179.020,5.329,148.629
C08915=1234.109,38.299,-43.119,-179.017,5.330,148.628
C08916=1234.103,38.548,-43.135,-179.015,5.330,148.627
C08917=1234.099,38.798,-43.151,-179.012,5.331,148.627
C08918=1234.094,39.047,-43.168,-179.009,5.331,148.626
C08919=1234.089,39.297,-43.184,-179.007,5.332,148.625
C08920=1234.084,39.546,-43.200,-179.005,5.332,148.625
C08921=1234.079,39.796,-43.216,-179.002,5.332,148.624
C08922=1234.074,40.045,-43.232,-178.999,5.333,148.623
C08923=1234.069,40.294,-43.249,-178.997,5.333,148.623
C08924=1234.064,40.543,-43.264,-178.994,5.334,148.622
C08925=1234.060,40.793,-43.281,-178.992,5.335,148.621
C08926=1234.054,41.042,-43.297,-178.989,5.334,148.621
C08927=1234.050,41.292,-43.313,-178.987,5.335,148.620
C08928=1234.045,41.541,-43.330,-178.985,5.336,148.620
C08929=1234.039,41.791,-43.346,-178.982,5.336,148.619
C08930=1234.034,42.040,-43.362,-178.979,5.337,148.618
C08931=1234.029,42.290,-43.378,-178.977,5.338,148.618
C08932=1234.024,42.539,-43.395,-178.974,5.338,148.617
C08933=1234.020,42.788,-43.411,-178.972,5.338,148.616
C08934=1234.015,43.038,-43.427,-178.969,5.338,148.616
C08935=1234.010,43.287,-43.444,-178.967,5.339,148.615
C08936=1234.005,43.537,-43.460,-178.964,5.340,148.614
C08937=1234.000,43.786,-43.476,-178.961,5.340,148.614
C08938=1233.995,44.036,-43.493,-178.959,5.341,148.613
C08939=1233.990,44.285,-43.509,-178.956,5.341,148.612
C08940=1233.985,44.535,-43.525,-178.954,5.341,148.612
C08941=1233.980,44.784,-43.542,-178.951,5.342,148.611
C08942=1233.975,45.033,-43.558,-178.949,5.342,148.610
C08943=1233.971,45.282,-43.575,-178.947,5.343,148.610
C08944=1233.965,45.532,-43.591,-178.944,5.344,148.609
C08945=1233.960,45.782,-43.608,-178.941,5.344,148.608
C08946=1233.955,46.030,-43.624,-178.939,5.345,148.608
C08947=1233.951,46.280,-43.641,-178.936,5.345,148.607
C08948=1233.946,46.530,-43.657,-178.934,5.345,148.606
C08949=1233.941,46.779,-43.673,-178.931,5.346,148.606
C08950=1233.936,47.029,-43.690,-178.929,5.346,148.605
C08951=1233.931,47.278,-43.707,-178.926,5.347,148.604
C08952=1233.926,47.527,-43.723,-178.924,5.347,148.604
C08953=1233.921,47.777,-43.739,-178.921,5.348,148.603
C08954=1233.915,48.026,-43.756,-178.918,5.349,148.602
C08955=1233.911,48.275,-43.773,-178.916,5.349,148.602
C08956=1233.906,48.525,-43.790,-178.914,5.349,148.601
C08957=1233.901,48.774,-43.806,-178.911,5.350,148.601
C08958=1233.897,49.023,-43.823,-178.909,5.350,148.600
C08959=1233.891,49.274,-43.839,-178.906,5.351,148.599
C08960=1233.886,49.522,-43.855,-178.903,5.352,148.599
C08961=1233.882,49.772,-43.872,-178.901,5.352,148.598
C08962=1233.877,50.022,-43.889,-178.898,5.353,148.597
C08963=1233.871,50.271,-43.906,-178.896,5.353,148.597
C08964=1233.867,50.520,-43.922,-178.893,5.354,148.596
C08965=1233.862,50.769,-43.939,-178.891,5.354,148.595
C08966=1233.857,51.019,-43.956,-178.888,5.354,148.595
C08967=1233.852,51.268,-43.973,-178.886,5.355,148.594
C08968=1233.848,51.518,-43.989,-178.883,5.356,148.593
C08969=1233.842,51.767,-44.006,-178.881,5.356,148.593
C08970=1233.837,52.016,-44.023,-178.878,5.357,148.592
C08971=1233.833,52.266,-44.039,-178.876,5.357,148.591
C08972=1233.827,52.515,-44.056,-178.873,5.358,148.591
C08973=1233.822,52.765,-44.072,-178.870,5.359,148.590
C08974=1233.818,53.014,-44.089,-178.868,5.359,148.589
C08975=1233.812,53.263,-44.106,-178.866,5.359,148.589
C08976=1233.808,53.513,-44.123,-178.863,5.359,148.588
C08977=1233.803,53.762,-44.139,-178.860,5.360,148.587
C08978=1233.798,54.012,-44.156,-178.858,5.361,148.587
C08979=1233.793,54.261,-44.173,-178.856,5.362,148.586
C08980=1233.788,54.510,-44.189,-178.853,5.362,148.586
C08981=1233.783,54.760,-44.207,-178.850,5.363,148.585
C08982=1233.778,55.008,-44.224,-178.848,5.363,148.584
C08983=1233.773,55.258,-44.241,-178.845,5.364,148.584
C08984=1233.768,55.527,-44.259,-178.842,5.364,148.583
C08985=1233.763,55.795,-44.276,-178.840,5.365,148.582
C08986=1233.757,56.064,-44.295,-178.837,5.366,148.582
C08987=1233.752,56.332,-44.313,-178.834,5.366,148.581
C08988=1233.747,56.582,-44.330,-178.832,5.367,148.580
C08989=1233.743,56.831,-44.347,-178.829,5.367,148.580
C08990=1233.738,57.080,-44.364,-178.827,5.368,148.579
C08991=1233.733,57.329,-44.381,-178.824,5.369,148.578
C08992=1233.727,57.579,-44.398,-178.822,5.368,148.578
C08993=1233.723,57.828,-44.415,-178.819,5.369,148.577
C08994=1233.718,58.078,-44.432,-178.817,5.369,148.576
C08995=1233.713,58.328,-44.449,-178.814,5.370,148.576
C08996=1233.708,58.576,-44.466,-178.812,5.371,148.575
C08997=1233.703,58.826,-44.483,-178.809,5.372,148.574
C08998=1233.699,59.075,-44.500,-178.807,5.372,148.574
C08999=1233.693,59.325,-44.517,-178.804,5.373,148.573
C09000=1233.688,59.574,-44.533,-178.801,5.373,148.572
C09001=1233.683,59.823,-44.551,-178.799,5.374,148.572
C09002=1233.679,60.072,-44.568,-178.796,5.374,148.571
C09003=1233.674,60.322,-44.585,-178.793,5.375,148.570
C09004=1233.669,60.572,-44.602,-178.791,5.376,148.570
C09005=1233.664,60.821,-44.620,-178.789,5.377,148.569
C09006=1233.659,61.070,-44.637,-178.786,5.377,148.569
C09007=1233.654,61.319,-44.653,-178.784,5.377,148.568
C09008=1233.649,61.569,-44.671,-178.781,5.378,148.567
C09009=1233.645,61.818,-44.688,-178.779,5.378,148.567
C09010=1233.639,62.068,-44.705,-178.776,5.379,148.566
C09011=1233.634,62.317,-44.721,-178.773,5.379,148.565
C09012=1233.629,62.566,-44.739,-178.771,5.380,148.565
C09013=1233.625,62.815,-44.756,-178.769,5.381,148.564
C09014=1233.620,63.065,-44.773,-178.766,5.381,148.564
C09015=1233.615,63.315,-44.791,-178.763,5.382,148.563
C09016=1233.610,63.564,-44.808,-178.761,5.383,148.562
C09017=1233.605,63.814,-44.825,-178.758,5.383,148.562
C09018=1233.600,64.062,-44.842,-178.755,5.384,148.561
C09019=1233.595,64.312,-44.860,-178.753,5.384,148.560
C09020=1233.590,64.561,-44.877,-178.751,5.385,148.560
C09021=1233.586,64.810,-44.894,-178.748,5.386,148.559
C09022=1233.581,65.060,-44.911,-178.745,5.386,148.559
C09023=1233.576,65.309,-44.928,-178.743,5.387,148.558
C09024=1233.571,65.559,-44.946,-178.740,5.388,148.557
C09025=1233.566,65.808,-44.963,-178.738,5.388,148.557
C09026=1233.562,66.057,-44.981,-178.735,5.388,148.556
C09027=1233.556,66.306,-44.998,-178.733,5.389,148.555
C09028=1233.551,66.556,-45.015,-178.731,5.390,148.555
C09029=1233.547,66.805,-45.032,-178.728,5.390,148.554
C09030=1233.541,67.055,-45.050,-178.725,5.391,148.553
C09031=1233.536,67.304,-45.068,-178.723,5.391,148.553
C09032=1233.532,67.554,-45.084,-178.720,5.392,148.552
C09033=1233.527,67.803,-45.102,-178.718,5.393,148.552
C09034=1233.522,68.053,-45.119,-178.715,5.393,148.551
C09035=1233.518,68.301,-45.137,-178.713,5.394,148.550
C09036=1233.512,68.551,-45.154,-178.710,5.395,148.550
C09037=1233.508,68.800,-45.172,-178.708,5.395,148.549
C09038=1233.502,69.050,-45.189,-178.705,5.396,148.548
C09039=1233.498,69.299,-45.207,-178.702,5.396,148.548
C09040=1233.493,69.549,-45.224,-178.700,5.397,148.547
C09041=1233.488,69.798,-45.242,-178.697,5.398,148.547
C09042=1233.483,70.046,-45.259,-178.695,5.398,148.546
C09043=1233.478,70.296,-45.276,-178.692,5.399,148.545
C09044=1233.473,70.545,-45.294,-178.690,5.400,148.545
C09045=1233.468,70.795,-45.312,-178.687,5.400,148.544
C09046=1233.464,71.044,-45.329,-178.685,5.401,148.544
C09047=1233.458,71.294,-45.346,-178.682,5.402,148.543
C09048=1233.454,71.543,-45.364,-178.680,5.402,148.542
C09049=1233.449,71.792,-45.382,-178.677,5.403,148.542
C09050=1233.443,72.042,-45.399,-178.674,5.404,148.541
C09051=1233.439,72.291,-45.417,-178.672,5.404,148.540
C09052=1233.434,72.540,-45.435,-178.670,5.405,148.540
C09053=1233.429,72.790,-45.452,-178.667,5.406,148.539
C09054=1233.424,73.039,-45.470,-178.664,5.406,148.539
C09055=1233.419,73.288,-45.488,-178.662,5.407,148.538
C09056=1233.415,73.537,-45.505,-178.659,5.407,148.537
C09057=1233.410,73.787,-45.523,-178.656,5.408,148.537
C09058=1233.405,74.036,-45.541,-178.654,5.409,148.536
C09059=1233.400,74.286,-45.558,-178.652,5.410,148.535
C09060=1233.395,74.535,-45.576,-178.649,5.410,148.535
C09061=1233.390,74.784,-45.594,-178.646,5.411,148.534
C09062=1233.385,75.033,-45.611,-178.644,5.411,148.533
C09063=1233.381,75.283,-45.629,-178.641,5.412,148.533
C09064=1233.376,75.532,-45.647,-178.639,5.413,148.532
C09065=1233.371,75.782,-45.665,-178.636,5.414,148.532
C09066=1233.366,76.031,-45.682,-178.634,5.414,148.531
C09067=1233.361,76.281,-45.700,-178.631,5.415,148.530
C09068=1233.356,76.530,-45.718,-178.629,5.415,148.530
C09069=1233.351,76.779,-45.736,-178.626,5.416,148.529
C09070=1233.346,77.028,-45.754,-178.624,5.417,148.529
C09071=1233.342,77.278,-45.771,-178.621,5.417,148.528
C09072=1233.337,77.527,-45.789,-178.618,5.418,148.527
C09073=1233.332,77.776,-45.807,-178.616,5.419,148.527
C09074=1233.327,78.025,-45.825,-178.614,5.420,148.526
C09075=1233.322,78.274,-45.843,-178.611,5.420,148.526
C09076=1233.317,78.523,-45.861,-178.608,5.421,148.525
C09077=1233.312,78.773,-45.878,-178.606,5.421,148.524
C09078=1233.307,79.022,-45.896,-178.603,5.422,148.524
C09079=1233.303,79.272,-45.914,-178.601,5.423,148.523
C09080=1233.298,79.521,-45.932,-178.598,5.424,148.523
C09081=1233.293,79.771,-45.950,-178.596,5.424,148.522
C09082=1233.288,80.020,-45.968,-178.593,5.425,148.521
C09083=1233.283,80.269,-45.986,-178.591,5.425,148.521
C09084=1233.278,80.518,-46.004,-178.588,5.426,148.520
C09085=1233.274,80.767,-46.022,-178.586,5.427,148.519
C09086=1233.268,81.017,-46.039,-178.583,5.428,148.519
C09087=1233.263,81.266,-46.057,-178.581,5.428,148.518
C09088=1233.258,81.535,-46.077,-178.578,5.429,148.518
C09089=1233.253,81.803,-46.096,-178.575,5.430,148.517
C09090=1233.248,82.071,-46.116,-178.572,5.431,148.516
C09091=1233.243,82.339,-46.135,-178.570,5.431,148.516
C09092=1233.238,82.590,-46.154,-178.567,5.432,148.515
C09093=1233.233,82.839,-46.172,-178.565,5.433,148.514
C09094=1233.228,83.088,-46.190,-178.562,5.434,148.514
C09095=1233.223,83.337,-46.208,-178.560,5.434,148.513
C09096=1233.218,83.586,-46.226,-178.557,5.435,148.512
C09097=1233.213,83.835,-46.244,-178.554,5.435,148.512
C09098=1233.209,84.085,-46.262,-178.552,5.436,148.511
C09099=1233.204,84.334,-46.280,-178.550,5.437,148.511
C09100=1233.199,84.584,-46.298,-178.547,5.438,148.510
C09101=1233.194,84.833,-46.316,-178.544,5.438,148.509
C09102=1233.189,85.082,-46.334,-178.542,5.440,148.509
C09103=1233.185,85.332,-46.352,-178.539,5.440,148.508
C09104=1233.180,85.581,-46.370,-178.536,5.441,148.508
C09105=1233.175,85.831,-46.389,-178.534,5.442,148.507
C09106=1233.170,86.079,-46.408,-178.531,5.442,148.506
C09107=1233.165,86.328,-46.426,-178.529,5.443,148.506
C09108=1233.161,86.578,-46.444,-178.526,5.444,148.505
C09109=1233.156,86.827,-46.462,-178.524,5.444,148.505
C09110=1233.151,87.076,-46.480,-178.521,5.445,148.504
C09111=1233.146,87.326,-46.498,-178.519,5.446,148.504
C09112=1233.140,87.575,-46.516,-178.516,5.447,148.503
C09113=1233.136,87.824,-46.536,-178.514,5.447,148.502
C09114=1233.131,88.074,-46.554,-178.511,5.448,148.502
C09115=1233.127,88.323,-46.571,-178.509,5.449,148.501
C09116=1233.122,88.572,-46.589,-178.506,5.449,148.501
C09117=1233.117,88.822,-46.608,-178.504,5.450,148.500
C09118=1233.112,89.071,-46.627,-178.501,5.451,148.499
C09119=1233.107,89.320,-46.645,-178.498,5.452,148.499
C09120=1233.102,89.569,-46.663,-178.496,5.453,148.498
C09121=1233.098,89.819,-46.681,-178.493,5.454,148.498
C09122=1233.093,90.068,-46.699,-178.491,5.454,148.497
C09123=1233.088,90.317,-46.719,-178.488,5.455,148.496
C09124=1233.083,90.566,-46.737,-178.486,5.456,148.496
C09125=1233.078,90.816,-46.755,-178.483,5.456,148.495
C09126=1233.074,91.065,-46.774,-178.481,5.457,148.495
C09127=1233.068,91.314,-46.792,-178.478,5.458,148.494
C09128=1233.064,91.564,-46.811,-178.476,5.459,148.493
C09129=1233.059,91.813,-46.829,-178.473,5.459,148.493
C09130=1233.054,92.062,-46.847,-178.471,5.460,148.492
C09131=1233.049,92.311,-46.866,-178.467,5.461,148.492
C09132=1233.044,92.561,-46.884,-178.465,5.462,148.491
C09133=1233.040,92.810,-46.903,-178.463,5.463,148.490
C09134=1233.034,93.059,-46.921,-178.460,5.463,148.490
